LIN {X 0,Y 432.697,Z 989.03,A -85,B 0,C 180,E1 8598.502,E2 8598.502} C_VEL
LIN {X 0,Y 432.77,Z 989.03,A -85,B 0,C 180,E1 8603.648,E2 8603.648} C_VEL
LIN {X 0,Y 432.907,Z 989.03,A -85,B 0,C 180,E1 8608.477,E2 8608.477} C_VEL
LIN {X 0,Y 433.07,Z 989.297,A -85,B 0,C 180,E1 8613.186,E2 8613.186} C_VEL
LIN {X 0,Y 443.785,Z 1017.541,A -85,B 0,C 180,E1 8615.048,E2 8615.048} C_VEL
LIN {X 0,Y 445.789,Z 1028.616,A -85,B 0,C 180,E1 8615.491,E2 8615.491} C_VEL
LIN {X 0,Y 445.07,Z 1060.716,A -85,B 0,C 180,E1 8616.568,E2 8616.568} C_VEL
LIN {X 0,Y 443.495,Z 1088.889,A -85,B 0,C 180,E1 8618.283,E2 8618.283} C_VEL
LIN {X 0,Y 441.306,Z 1114.853,A -85,B 0,C 180,E1 8620.732,E2 8620.732} C_VEL
LIN {X 0,Y 439.12,Z 1136.774,A -85,B 0,C 180,E1 8623.787,E2 8623.787} C_VEL
LIN {X 0,Y 437.236,Z 1152.919,A -85,B 0,C 180,E1 8627.037,E2 8627.037} C_VEL
LIN {X 0,Y 436.045,Z 1164.999,A -85,B 0,C 180,E1 8630.715,E2 8630.715} C_VEL
LIN {X 0,Y 435.323,Z 1172.825,A -85,B 0,C 180,E1 8635.028,E2 8635.028} C_VEL
LIN {X 0,Y 435.121,Z 1174.716,A -85,B 0,C 180,E1 8638.012,E2 8638.012} C_VEL
LIN {X 0,Y 435.207,Z 1172.894,A -85,B 0,C 180,E1 8641.987,E2 8641.987} C_VEL
LIN {X 0,Y 435.483,Z 1166.041,A -85,B 0,C 180,E1 8645.966,E2 8645.966} C_VEL
LIN {X 0,Y 436.346,Z 1153.47,A -85,B 0,C 180,E1 8649.956,E2 8649.956} C_VEL
LIN {X 0,Y 437.774,Z 1136.478,A -85,B 0,C 180,E1 8653.453,E2 8653.453} C_VEL
LIN {X 0,Y 439.79,Z 1114.572,A -85,B 0,C 180,E1 8656.571,E2 8656.571} C_VEL
LIN {X 0,Y 442.047,Z 1087.996,A -85,B 0,C 180,E1 8659.181,E2 8659.181} C_VEL
LIN {X 0,Y 443.923,Z 1058.883,A -85,B 0,C 180,E1 8661.067,E2 8661.067} C_VEL
LIN {X 0,Y 445.087,Z 1027.458,A -85,B 0,C 180,E1 8662.249,E2 8662.249} C_VEL
LIN {X 0,Y 442.129,Z 1014.96,A -85,B 0,C 180,E1 8662.7,E2 8662.7} C_VEL
LIN {X 0,Y 433.211,Z 989.03,A -85,B 0,C 180,E1 8663.83,E2 8663.83} C_VEL
LIN {X 0,Y 432.895,Z 989.03,A -85,B 0,C 180,E1 8669.36,E2 8669.36} C_VEL
LIN {X 0,Y 432.823,Z 989.03,A -85,B 0,C 180,E1 8673.904,E2 8673.904} C_VEL
LIN {X 0,Y 432.669,Z 989.03,A -85,B 0,C 180,E1 8679.881,E2 8679.881} C_VEL
LIN {X 0,Y 432.821,Z 989.03,A -85,B 0,C 180,E1 8687.064,E2 8687.064} C_VEL
LIN {X 0,Y 433.004,Z 989.789,A -85,B 0,C 180,E1 8692.927,E2 8692.927} C_VEL
LIN {X 0,Y 456.109,Z 1039.383,A -85,B 0,C 180,E1 8696.121,E2 8696.121} C_VEL
LIN {X 0,Y 454.129,Z 1077.382,A -85,B 0,C 180,E1 8697.482,E2 8697.482} C_VEL
LIN {X 0,Y 450.882,Z 1111.659,A -85,B 0,C 180,E1 8699.45,E2 8699.45} C_VEL
LIN {X 0,Y 446.779,Z 1144.475,A -85,B 0,C 180,E1 8702.186,E2 8702.186} C_VEL
LIN {X 0,Y 442.832,Z 1172.505,A -85,B 0,C 180,E1 8705.44,E2 8705.44} C_VEL
LIN {X 0,Y 439.203,Z 1197.466,A -85,B 0,C 180,E1 8709.375,E2 8709.375} C_VEL
LIN {X 0,Y 436.454,Z 1218.293,A -85,B 0,C 180,E1 8713.938,E2 8713.938} C_VEL
LIN {X 0,Y 435.007,Z 1232.645,A -85,B 0,C 180,E1 8718.49,E2 8718.49} C_VEL
LIN {X 0,Y 434.441,Z 1241.786,A -85,B 0,C 180,E1 8723.013,E2 8723.013} C_VEL
LIN {X 0,Y 434.17,Z 1246.568,A -85,B 0,C 180,E1 8728.004,E2 8728.004} C_VEL
LIN {X 0,Y 434.304,Z 1246.516,A -85,B 0,C 180,E1 8731.987,E2 8731.987} C_VEL
LIN {X 0,Y 434.395,Z 1241.668,A -85,B 0,C 180,E1 8736.98,E2 8736.98} C_VEL
LIN {X 0,Y 435.171,Z 1231.159,A -85,B 0,C 180,E1 8742.005,E2 8742.005} C_VEL
LIN {X 0,Y 436.864,Z 1214.961,A -85,B 0,C 180,E1 8746.812,E2 8746.812} C_VEL
LIN {X 0,Y 439.667,Z 1194.228,A -85,B 0,C 180,E1 8751.12,E2 8751.12} C_VEL
LIN {X 0,Y 443.383,Z 1168.758,A -85,B 0,C 180,E1 8754.97,E2 8754.97} C_VEL
LIN {X 0,Y 447.385,Z 1139.749,A -85,B 0,C 180,E1 8758.175,E2 8758.175} C_VEL
LIN {X 0,Y 451.302,Z 1107.239,A -85,B 0,C 180,E1 8760.762,E2 8760.762} C_VEL
LIN {X 0,Y 454.599,Z 1071.466,A -85,B 0,C 180,E1 8762.694,E2 8762.694} C_VEL
LIN {X 0,Y 455.862,Z 1038.327,A -85,B 0,C 180,E1 8763.838,E2 8763.838} C_VEL
LIN {X 0,Y 436.175,Z 997.068,A -85,B 0,C 180,E1 8766.511,E2 8766.511} C_VEL
LIN {X 0,Y 432.88,Z 989.03,A -85,B 0,C 180,E1 8767.031,E2 8767.031} C_VEL
LIN {X 0,Y 432.718,Z 989.03,A -85,B 0,C 180,E1 8774.22,E2 8774.22} C_VEL
LIN {X 0,Y 432.769,Z 989.03,A -85,B 0,C 180,E1 8780.091,E2 8780.091} C_VEL
LIN {X 0,Y 432.886,Z 989.03,A -85,B 0,C 180,E1 8786.781,E2 8786.781} C_VEL
LIN {X 0,Y 433.033,Z 989.03,A -85,B 0,C 180,E1 8793.064,E2 8793.064} C_VEL
LIN {X 0,Y 433.316,Z 989.03,A -85,B 0,C 180,E1 8800.09,E2 8800.09} C_VEL
LIN {X 0,Y 433.537,Z 989.03,A -85,B 0,C 180,E1 8805.899,E2 8805.899} C_VEL
LIN {X 0,Y 433.62,Z 989.03,A -85,B 0,C 180,E1 8812.633,E2 8812.633} C_VEL
LIN {X 0,Y 433.826,Z 989.03,A -85,B 0,C 180,E1 8818.007,E2 8818.007} C_VEL
LIN {X 0,Y 433.765,Z 989.03,A -85,B 0,C 180,E1 8823.99,E2 8823.99} C_VEL
LIN {X 0,Y 433.535,Z 989.03,A -85,B 0,C 180,E1 8830.022,E2 8830.022} C_VEL
LIN {X 0,Y 433.346,Z 989.03,A -85,B 0,C 180,E1 8836.175,E2 8836.175} C_VEL
LIN {X 0,Y 433.179,Z 989.03,A -85,B 0,C 180,E1 8842.531,E2 8842.531} C_VEL
LIN {X 0,Y 432.896,Z 989.03,A -85,B 0,C 180,E1 8849.376,E2 8849.376} C_VEL
LIN {X 0,Y 432.837,Z 989.03,A -85,B 0,C 180,E1 8853.903,E2 8853.903} C_VEL
LIN {X 0,Y 432.775,Z 989.03,A -85,B 0,C 180,E1 8859.91,E2 8859.91} C_VEL
LIN {X 0,Y 432.855,Z 989.105,A -85,B 0,C 180,E1 8865.604,E2 8865.604} C_VEL
LIN {X 0,Y 442.678,Z 1017.502,A -85,B 0,C 180,E1 8868.683,E2 8868.683} C_VEL
LIN {X 0,Y 458.724,Z 1050.911,A -85,B 0,C 180,E1 8870.893,E2 8870.893} C_VEL
LIN {X 0,Y 460.741,Z 1053.948,A -85,B 0,C 180,E1 8871.137,E2 8871.137} C_VEL
LIN {X 0,Y 458.124,Z 1095.324,A -85,B 0,C 180,E1 8872.358,E2 8872.358} C_VEL
LIN {X 0,Y 454.341,Z 1134.437,A -85,B 0,C 180,E1 8874.243,E2 8874.243} C_VEL
LIN {X 0,Y 449.841,Z 1172.08,A -85,B 0,C 180,E1 8876.863,E2 8876.863} C_VEL
LIN {X 0,Y 446.664,Z 1196.79,A -85,B 0,C 180,E1 8879.099,E2 8879.099} C_VEL
LIN {X 0,Y 441.188,Z 1210.269,A -85,B 0,C 180,E1 8880.368,E2 8880.368} C_VEL
LIN {X 0,Y 435.677,Z 1223.042,A -85,B 0,C 180,E1 8881.762,E2 8881.762} C_VEL
LIN {X 0,Y 431.796,Z 1251.772,A -85,B 0,C 180,E1 8886.033,E2 8886.033} C_VEL
LIN {X 0,Y 428.851,Z 1276.693,A -85,B 0,C 180,E1 8891.009,E2 8891.009} C_VEL
LIN {X 0,Y 427.165,Z 1294.995,A -85,B 0,C 180,E1 8896.163,E2 8896.163} C_VEL
LIN {X 0,Y 426.423,Z 1306.284,A -85,B 0,C 180,E1 8900.841,E2 8900.841} C_VEL
LIN {X 0,Y 426.181,Z 1310.937,A -85,B 0,C 180,E1 8903.906,E2 8903.906} C_VEL
LIN {X 0,Y 426.118,Z 1314.097,A -85,B 0,C 180,E1 8907.974,E2 8907.974} C_VEL
LIN {X 0,Y 426.159,Z 1314.101,A -85,B 0,C 180,E1 8912.033,E2 8912.033} C_VEL
LIN {X 0,Y 426.297,Z 1309.951,A -85,B 0,C 180,E1 8916.886,E2 8916.886} C_VEL
LIN {X 0,Y 426.714,Z 1300.562,A -85,B 0,C 180,E1 8921.737,E2 8921.737} C_VEL
LIN {X 0,Y 427.905,Z 1286.255,A -85,B 0,C 180,E1 8926.391,E2 8926.391} C_VEL
LIN {X 0,Y 429.839,Z 1266.674,A -85,B 0,C 180,E1 8930.887,E2 8930.887} C_VEL
LIN {X 0,Y 432.863,Z 1239.391,A -85,B 0,C 180,E1 8935.454,E2 8935.454} C_VEL
LIN {X 0,Y 436.533,Z 1207.714,A -85,B 0,C 180,E1 8939.357,E2 8939.357} C_VEL
LIN {X 0,Y 440.383,Z 1171.631,A -85,B 0,C 180,E1 8942.668,E2 8942.668} C_VEL
LIN {X 0,Y 444.264,Z 1131,A -85,B 0,C 180,E1 8945.396,E2 8945.396} C_VEL
LIN {X 0,Y 447.832,Z 1087.494,A -85,B 0,C 180,E1 8947.417,E2 8947.417} C_VEL
LIN {X 0,Y 449.457,Z 1053.468,A -85,B 0,C 180,E1 8948.495,E2 8948.495} C_VEL
LIN {X 0,Y 439.336,Z 1031.663,A -85,B 0,C 180,E1 8949.877,E2 8949.877} C_VEL
LIN {X 0,Y 429.889,Z 1001.599,A -85,B 0,C 180,E1 8951.62,E2 8951.62} C_VEL
LIN {X 0,Y 424.951,Z 989.03,A -85,B 0,C 180,E1 8952.743,E2 8952.743} C_VEL
LIN {X 0,Y 424.781,Z 989.03,A -85,B 0,C 180,E1 8960.252,E2 8960.252} C_VEL
LIN {X 0,Y 424.859,Z 989.03,A -85,B 0,C 180,E1 8965.371,E2 8965.371} C_VEL
LIN {X 0,Y 425.05,Z 989.03,A -85,B 0,C 180,E1 8971.942,E2 8971.942} C_VEL
LIN {X 0,Y 425.08,Z 989.609,A -85,B 0,C 180,E1 8972.308,E2 8972.308} C_VEL
LIN {X 0,Y 435.465,Z 1014.789,A -85,B 0,C 180,E1 8974.299,E2 8974.299} C_VEL
LIN {X 0,Y 438.864,Z 1029.178,A -85,B 0,C 180,E1 8975.006,E2 8975.006} C_VEL
LIN {X 0,Y 438.027,Z 1062.901,A -85,B 0,C 180,E1 8976.168,E2 8976.168} C_VEL
LIN {X 0,Y 436.35,Z 1090.736,A -85,B 0,C 180,E1 8977.91,E2 8977.91} C_VEL
LIN {X 0,Y 434.06,Z 1116.2,A -85,B 0,C 180,E1 8980.354,E2 8980.354} C_VEL
LIN {X 0,Y 431.726,Z 1138.391,A -85,B 0,C 180,E1 8983.502,E2 8983.502} C_VEL
LIN {X 0,Y 429.681,Z 1154.456,A -85,B 0,C 180,E1 8986.805,E2 8986.805} C_VEL
LIN {X 0,Y 428.41,Z 1166.411,A -85,B 0,C 180,E1 8990.524,E2 8990.524} C_VEL
LIN {X 0,Y 427.732,Z 1173.018,A -85,B 0,C 180,E1 8993.924,E2 8993.924} C_VEL
LIN {X 0,Y 427.362,Z 1176.103,A -85,B 0,C 180,E1 8997.976,E2 8997.976} C_VEL
LIN {X 0,Y 427.447,Z 1174.222,A -85,B 0,C 180,E1 9002.023,E2 9002.023} C_VEL
LIN {X 0,Y 427.731,Z 1167.313,A -85,B 0,C 180,E1 9006.075,E2 9006.075} C_VEL
LIN {X 0,Y 428.678,Z 1154.67,A -85,B 0,C 180,E1 9010.136,E2 9010.136} C_VEL
LIN {X 0,Y 430.176,Z 1137.616,A -85,B 0,C 180,E1 9013.696,E2 9013.696} C_VEL
LIN {X 0,Y 432.314,Z 1115.636,A -85,B 0,C 180,E1 9016.866,E2 9016.866} C_VEL
LIN {X 0,Y 434.667,Z 1088.998,A -85,B 0,C 180,E1 9019.519,E2 9019.519} C_VEL
LIN {X 0,Y 436.668,Z 1058.992,A -85,B 0,C 180,E1 9021.478,E2 9021.478} C_VEL
LIN {X 0,Y 437.856,Z 1027.198,A -85,B 0,C 180,E1 9022.669,E2 9022.669} C_VEL
LIN {X 0,Y 425.204,Z 989.03,A -85,B 0,C 180,E1 9024.362,E2 9024.362} C_VEL
LIN {X 0,Y 424.94,Z 989.03,A -85,B 0,C 180,E1 9031.531,E2 9031.531} C_VEL
LIN {X 0,Y 424.741,Z 989.03,A -85,B 0,C 180,E1 9038.583,E2 9038.583} C_VEL
LIN {X 0,Y 424.87,Z 989.03,A -85,B 0,C 180,E1 9045.259,E2 9045.259} C_VEL
LIN {X 0,Y 424.987,Z 989.187,A -85,B 0,C 180,E1 9052.082,E2 9052.082} C_VEL
LIN {X 0,Y 431.957,Z 1003.724,A -85,B 0,C 180,E1 9053.108,E2 9053.108} C_VEL
LIN {X 0,Y 449.723,Z 1042.379,A -85,B 0,C 180,E1 9055.652,E2 9055.652} C_VEL
LIN {X 0,Y 447.403,Z 1079.179,A -85,B 0,C 180,E1 9056.998,E2 9056.998} C_VEL
LIN {X 0,Y 443.964,Z 1113.426,A -85,B 0,C 180,E1 9059.015,E2 9059.015} C_VEL
LIN {X 0,Y 439.582,Z 1146.278,A -85,B 0,C 180,E1 9061.83,E2 9061.83} C_VEL
LIN {X 0,Y 435.379,Z 1174.63,A -85,B 0,C 180,E1 9065.219,E2 9065.219} C_VEL
LIN {X 0,Y 431.559,Z 1199.462,A -85,B 0,C 180,E1 9069.261,E2 9069.261} C_VEL
LIN {X 0,Y 428.808,Z 1218.892,A -85,B 0,C 180,E1 9073.644,E2 9073.644} C_VEL
LIN {X 0,Y 427.245,Z 1233.244,A -85,B 0,C 180,E1 9078.278,E2 9078.278} C_VEL
LIN {X 0,Y 426.584,Z 1242.464,A -85,B 0,C 180,E1 9082.936,E2 9082.936} C_VEL
LIN {X 0,Y 426.293,Z 1247.169,A -85,B 0,C 180,E1 9087.967,E2 9087.967} C_VEL
LIN {X 0,Y 426.425,Z 1247.118,A -85,B 0,C 180,E1 9092.024,E2 9092.024} C_VEL
LIN {X 0,Y 426.543,Z 1242.349,A -85,B 0,C 180,E1 9097.056,E2 9097.056} C_VEL
LIN {X 0,Y 427.266,Z 1233.044,A -85,B 0,C 180,E1 9101.713,E2 9101.713} C_VEL
LIN {X 0,Y 428.955,Z 1218.59,A -85,B 0,C 180,E1 9106.342,E2 9106.342} C_VEL
LIN {X 0,Y 431.839,Z 1197.629,A -85,B 0,C 180,E1 9110.985,E2 9110.985} C_VEL
LIN {X 0,Y 435.654,Z 1172.61,A -85,B 0,C 180,E1 9114.972,E2 9114.972} C_VEL
LIN {X 0,Y 440.031,Z 1143.028,A -85,B 0,C 180,E1 9118.409,E2 9118.409} C_VEL
LIN {X 0,Y 444.192,Z 1110.636,A -85,B 0,C 180,E1 9121.091,E2 9121.091} C_VEL
LIN {X 0,Y 447.715,Z 1075.651,A -85,B 0,C 180,E1 9123.072,E2 9123.072} C_VEL
LIN {X 0,Y 449.208,Z 1040.792,A -85,B 0,C 180,E1 9124.351,E2 9124.351} C_VEL
LIN {X 0,Y 430.884,Z 1001.912,A -85,B 0,C 180,E1 9126.942,E2 9126.942} C_VEL
LIN {X 0,Y 424.926,Z 989.03,A -85,B 0,C 180,E1 9127.915,E2 9127.915} C_VEL
LIN {X 0,Y 424.845,Z 989.03,A -85,B 0,C 180,E1 9135.262,E2 9135.262} C_VEL
LIN {X 0,Y 424.883,Z 989.03,A -85,B 0,C 180,E1 9141.38,E2 9141.38} C_VEL
LIN {X 0,Y 424.936,Z 989.03,A -85,B 0,C 180,E1 9148.455,E2 9148.455} C_VEL
LIN {X 0,Y 425.168,Z 989.03,A -85,B 0,C 180,E1 9154.794,E2 9154.794} C_VEL
LIN {X 0,Y 425.405,Z 989.03,A -85,B 0,C 180,E1 9161.384,E2 9161.384} C_VEL
LIN {X 0,Y 425.664,Z 989.03,A -85,B 0,C 180,E1 9167.72,E2 9167.72} C_VEL
LIN {X 0,Y 425.813,Z 989.03,A -85,B 0,C 180,E1 9173.898,E2 9173.898} C_VEL
LIN {X 0,Y 426.058,Z 989.03,A -85,B 0,C 180,E1 9180,E2 9180} C_VEL
LIN {X 0,Y 425.737,Z 989.03,A -85,B 0,C 180,E1 9187.064,E2 9187.064} C_VEL
LIN {X 0,Y 425.577,Z 989.03,A -85,B 0,C 180,E1 9192.283,E2 9192.283} C_VEL
LIN {X 0,Y 425.328,Z 989.03,A -85,B 0,C 180,E1 9198.621,E2 9198.621} C_VEL
LIN {X 0,Y 425.133,Z 989.03,A -85,B 0,C 180,E1 9205.209,E2 9205.209} C_VEL
LIN {X 0,Y 424.909,Z 989.03,A -85,B 0,C 180,E1 9212.187,E2 9212.187} C_VEL
LIN {X 0,Y 424.887,Z 989.03,A -85,B 0,C 180,E1 9218.621,E2 9218.621} C_VEL
LIN {X 0,Y 424.923,Z 989.717,A -85,B 0,C 180,E1 9224.886,E2 9224.886} C_VEL
LIN {X 0,Y 434.69,Z 1016.637,A -85,B 0,C 180,E1 9227.89,E2 9227.89} C_VEL
LIN {X 0,Y 453.005,Z 1055.473,A -85,B 0,C 180,E1 9230.511,E2 9230.511} C_VEL
LIN {X 0,Y 454.078,Z 1059.186,A -85,B 0,C 180,E1 9230.7,E2 9230.7} C_VEL
LIN {X 0,Y 450.861,Z 1100.733,A -85,B 0,C 180,E1 9232.056,E2 9232.056} C_VEL
LIN {X 0,Y 446.505,Z 1141.499,A -85,B 0,C 180,E1 9234.201,E2 9234.201} C_VEL
LIN {X 0,Y 441.692,Z 1178.777,A -85,B 0,C 180,E1 9237.013,E2 9237.013} C_VEL
LIN {X 0,Y 436.921,Z 1213.948,A -85,B 0,C 180,E1 9240.629,E2 9240.629} C_VEL
LIN {X 0,Y 435.677,Z 1223.042,A -85,B 0,C 180,E1 9241.762,E2 9241.762} C_VEL
LIN {X 0,Y 430.057,Z 1235.144,A -85,B 0,C 180,E1 9243.282,E2 9243.282} C_VEL
LIN {X 0,Y 424.722,Z 1246.437,A -85,B 0,C 180,E1 9244.928,E2 9244.928} C_VEL
LIN {X 0,Y 421.591,Z 1270.624,A -85,B 0,C 180,E1 9249.578,E2 9249.578} C_VEL
LIN {X 0,Y 419.716,Z 1289.061,A -85,B 0,C 180,E1 9254.36,E2 9254.36} C_VEL
LIN {X 0,Y 418.78,Z 1301.967,A -85,B 0,C 180,E1 9259.099,E2 9259.099} C_VEL
LIN {X 0,Y 418.338,Z 1309.955,A -85,B 0,C 180,E1 9263.791,E2 9263.791} C_VEL
LIN {X 0,Y 418.241,Z 1313.389,A -85,B 0,C 180,E1 9267.936,E2 9267.936} C_VEL
LIN {X 0,Y 418.281,Z 1313.385,A -85,B 0,C 180,E1 9272.072,E2 9272.072} C_VEL
LIN {X 0,Y 418.395,Z 1309.9,A -85,B 0,C 180,E1 9276.216,E2 9276.216} C_VEL
LIN {X 0,Y 418.831,Z 1300.391,A -85,B 0,C 180,E1 9281.434,E2 9281.434} C_VEL
LIN {X 0,Y 419.957,Z 1286.383,A -85,B 0,C 180,E1 9286.174,E2 9286.174} C_VEL
LIN {X 0,Y 421.967,Z 1266.202,A -85,B 0,C 180,E1 9290.959,E2 9290.959} C_VEL
LIN {X 0,Y 424.771,Z 1241.45,A -85,B 0,C 180,E1 9295.238,E2 9295.238} C_VEL
LIN {X 0,Y 428.288,Z 1211.677,A -85,B 0,C 180,E1 9299.114,E2 9299.114} C_VEL
LIN {X 0,Y 432.282,Z 1176.111,A -85,B 0,C 180,E1 9302.591,E2 9302.591} C_VEL
LIN {X 0,Y 436.468,Z 1135.133,A -85,B 0,C 180,E1 9305.529,E2 9305.529} C_VEL
LIN {X 0,Y 440.479,Z 1090.079,A -85,B 0,C 180,E1 9307.767,E2 9307.767} C_VEL
LIN {X 0,Y 442.462,Z 1056.367,A -85,B 0,C 180,E1 9308.923,E2 9308.923} C_VEL
LIN {X 0,Y 432.925,Z 1034.002,A -85,B 0,C 180,E1 9310.416,E2 9310.416} C_VEL
LIN {X 0,Y 423.891,Z 1004.177,A -85,B 0,C 180,E1 9312.262,E2 9312.262} C_VEL
LIN {X 0,Y 418.544,Z 993.693,A -85,B 0,C 180,E1 9313.357,E2 9313.357} C_VEL
LIN {X 0,Y 416.956,Z 989.03,A -85,B 0,C 180,E1 9313.91,E2 9313.91} C_VEL
LIN {X 0,Y 416.829,Z 989.03,A -85,B 0,C 180,E1 9319.494,E2 9319.494} C_VEL
LIN {X 0,Y 416.916,Z 989.03,A -85,B 0,C 180,E1 9326.363,E2 9326.363} C_VEL
LIN {X 0,Y 417.138,Z 989.03,A -85,B 0,C 180,E1 9331.219,E2 9331.219} C_VEL
LIN {X 0,Y 427.512,Z 1013.324,A -85,B 0,C 180,E1 9333.524,E2 9333.524} C_VEL
LIN {X 0,Y 432.04,Z 1030.019,A -85,B 0,C 180,E1 9334.495,E2 9334.495} C_VEL
LIN {X 0,Y 431.091,Z 1064.164,A -85,B 0,C 180,E1 9335.697,E2 9335.697} C_VEL
LIN {X 0,Y 429.277,Z 1092.763,A -85,B 0,C 180,E1 9337.526,E2 9337.526} C_VEL
LIN {X 0,Y 426.758,Z 1118.671,A -85,B 0,C 180,E1 9340.089,E2 9340.089} C_VEL
LIN {X 0,Y 424.327,Z 1140.066,A -85,B 0,C 180,E1 9343.206,E2 9343.206} C_VEL
LIN {X 0,Y 422.143,Z 1156.036,A -85,B 0,C 180,E1 9346.565,E2 9346.565} C_VEL
LIN {X 0,Y 420.754,Z 1167.929,A -85,B 0,C 180,E1 9350.35,E2 9350.35} C_VEL
LIN {X 0,Y 420.03,Z 1174.471,A -85,B 0,C 180,E1 9353.813,E2 9353.813} C_VEL
LIN {X 0,Y 419.606,Z 1177.5,A -85,B 0,C 180,E1 9357.939,E2 9357.939} C_VEL
LIN {X 0,Y 419.679,Z 1175.549,A -85,B 0,C 180,E1 9362.06,E2 9362.06} C_VEL
LIN {X 0,Y 419.988,Z 1168.561,A -85,B 0,C 180,E1 9366.187,E2 9366.187} C_VEL
LIN {X 0,Y 420.994,Z 1155.832,A -85,B 0,C 180,E1 9370.323,E2 9370.323} C_VEL
LIN {X 0,Y 422.574,Z 1138.687,A -85,B 0,C 180,E1 9373.947,E2 9373.947} C_VEL
LIN {X 0,Y 424.921,Z 1115.581,A -85,B 0,C 180,E1 9377.301,E2 9377.301} C_VEL
LIN {X 0,Y 427.441,Z 1088.267,A -85,B 0,C 180,E1 9379.997,E2 9379.997} C_VEL
LIN {X 0,Y 429.389,Z 1059.763,A -85,B 0,C 180,E1 9381.861,E2 9381.861} C_VEL
LIN {X 0,Y 430.389,Z 1026.985,A -85,B 0,C 180,E1 9383.107,E2 9383.107} C_VEL
LIN {X 0,Y 417.283,Z 989.03,A -85,B 0,C 180,E1 9384.893,E2 9384.893} C_VEL
LIN {X 0,Y 417.025,Z 989.03,A -85,B 0,C 180,E1 9390.435,E2 9390.435} C_VEL
LIN {X 0,Y 416.847,Z 989.03,A -85,B 0,C 180,E1 9397.202,E2 9397.202} C_VEL
LIN {X 0,Y 416.84,Z 989.03,A -85,B 0,C 180,E1 9403.605,E2 9403.605} C_VEL
LIN {X 0,Y 416.976,Z 989.03,A -85,B 0,C 180,E1 9410.496,E2 9410.496} C_VEL
LIN {X 0,Y 417.012,Z 989.033,A -85,B 0,C 180,E1 9411.209,E2 9411.209} C_VEL
LIN {X 0,Y 421.339,Z 998.671,A -85,B 0,C 180,E1 9411.893,E2 9411.893} C_VEL
LIN {X 0,Y 441.202,Z 1039.657,A -85,B 0,C 180,E1 9414.786,E2 9414.786} C_VEL
LIN {X 0,Y 443.045,Z 1046.799,A -85,B 0,C 180,E1 9415.186,E2 9415.186} C_VEL
LIN {X 0,Y 440.312,Z 1084.785,A -85,B 0,C 180,E1 9416.679,E2 9416.679} C_VEL
LIN {X 0,Y 436.489,Z 1119.573,A -85,B 0,C 180,E1 9418.902,E2 9418.902} C_VEL
LIN {X 0,Y 432.046,Z 1150.522,A -85,B 0,C 180,E1 9421.72,E2 9421.72} C_VEL
LIN {X 0,Y 427.643,Z 1178.421,A -85,B 0,C 180,E1 9425.222,E2 9425.222} C_VEL
LIN {X 0,Y 423.67,Z 1202.649,A -85,B 0,C 180,E1 9429.402,E2 9429.402} C_VEL
LIN {X 0,Y 420.924,Z 1221.353,A -85,B 0,C 180,E1 9433.864,E2 9433.864} C_VEL
LIN {X 0,Y 419.347,Z 1235.118,A -85,B 0,C 180,E1 9438.58,E2 9438.58} C_VEL
LIN {X 0,Y 418.641,Z 1244.422,A -85,B 0,C 180,E1 9443.788,E2 9443.788} C_VEL
LIN {X 0,Y 418.415,Z 1247.77,A -85,B 0,C 180,E1 9447.929,E2 9447.929} C_VEL
LIN {X 0,Y 418.545,Z 1247.72,A -85,B 0,C 180,E1 9452.062,E2 9452.062} C_VEL
LIN {X 0,Y 418.678,Z 1243.217,A -85,B 0,C 180,E1 9457.002,E2 9457.002} C_VEL
LIN {X 0,Y 419.504,Z 1233.648,A -85,B 0,C 180,E1 9461.933,E2 9461.933} C_VEL
LIN {X 0,Y 421.281,Z 1219.199,A -85,B 0,C 180,E1 9466.648,E2 9466.648} C_VEL
LIN {X 0,Y 424.36,Z 1198.426,A -85,B 0,C 180,E1 9471.335,E2 9471.335} C_VEL
LIN {X 0,Y 428.369,Z 1173.656,A -85,B 0,C 180,E1 9475.359,E2 9475.359} C_VEL
LIN {X 0,Y 433.085,Z 1143.62,A -85,B 0,C 180,E1 9478.908,E2 9478.908} C_VEL
LIN {X 0,Y 437.471,Z 1111.065,A -85,B 0,C 180,E1 9481.635,E2 9481.635} C_VEL
LIN {X 0,Y 441.144,Z 1075.926,A -85,B 0,C 180,E1 9483.645,E2 9483.645} C_VEL
LIN {X 0,Y 442.733,Z 1043.418,A -85,B 0,C 180,E1 9484.858,E2 9484.858} C_VEL
LIN {X 0,Y 424.334,Z 1004.19,A -85,B 0,C 180,E1 9487.572,E2 9487.572} C_VEL
LIN {X 0,Y 417.022,Z 990.228,A -85,B 0,C 180,E1 9488.665,E2 9488.665} C_VEL
LIN {X 0,Y 416.949,Z 989.03,A -85,B 0,C 180,E1 9488.725,E2 9488.725} C_VEL
LIN {X 0,Y 416.877,Z 989.03,A -85,B 0,C 180,E1 9496.378,E2 9496.378} C_VEL
LIN {X 0,Y 417.014,Z 989.03,A -85,B 0,C 180,E1 9502.754,E2 9502.754} C_VEL
LIN {X 0,Y 417.058,Z 989.03,A -85,B 0,C 180,E1 9510.265,E2 9510.265} C_VEL
LIN {X 0,Y 417.304,Z 989.03,A -85,B 0,C 180,E1 9516.563,E2 9516.563} C_VEL
LIN {X 0,Y 417.566,Z 989.03,A -85,B 0,C 180,E1 9523.197,E2 9523.197} C_VEL
LIN {X 0,Y 417.761,Z 989.03,A -85,B 0,C 180,E1 9529.596,E2 9529.596} C_VEL
LIN {X 0,Y 417.998,Z 989.03,A -85,B 0,C 180,E1 9535.86,E2 9535.86} C_VEL
LIN {X 0,Y 418.182,Z 989.03,A -85,B 0,C 180,E1 9542.068,E2 9542.068} C_VEL
LIN {X 0,Y 417.79,Z 989.03,A -85,B 0,C 180,E1 9548.307,E2 9548.307} C_VEL
LIN {X 0,Y 417.539,Z 989.03,A -85,B 0,C 180,E1 9554.654,E2 9554.654} C_VEL
LIN {X 0,Y 417.337,Z 989.03,A -85,B 0,C 180,E1 9561.197,E2 9561.197} C_VEL
LIN {X 0,Y 417.067,Z 989.03,A -85,B 0,C 180,E1 9568.057,E2 9568.057} C_VEL
LIN {X 0,Y 416.946,Z 989.03,A -85,B 0,C 180,E1 9575.384,E2 9575.384} C_VEL
LIN {X 0,Y 416.921,Z 989.03,A -85,B 0,C 180,E1 9580.653,E2 9580.653} C_VEL
LIN {X 0,Y 416.937,Z 989.221,A -85,B 0,C 180,E1 9584.043,E2 9584.043} C_VEL
LIN {X 0,Y 426.396,Z 1015.45,A -85,B 0,C 180,E1 9587.037,E2 9587.037} C_VEL
LIN {X 0,Y 447.39,Z 1061.599,A -85,B 0,C 180,E1 9590.201,E2 9590.201} C_VEL
LIN {X 0,Y 443.922,Z 1102.643,A -85,B 0,C 180,E1 9591.607,E2 9591.607} C_VEL
LIN {X 0,Y 439.459,Z 1141.866,A -85,B 0,C 180,E1 9593.742,E2 9593.742} C_VEL
LIN {X 0,Y 434.489,Z 1178.285,A -85,B 0,C 180,E1 9596.555,E2 9596.555} C_VEL
LIN {X 0,Y 429.614,Z 1212.439,A -85,B 0,C 180,E1 9600.116,E2 9600.116} C_VEL
LIN {X 0,Y 425.114,Z 1243.426,A -85,B 0,C 180,E1 9604.439,E2 9604.439} C_VEL
LIN {X 0,Y 424.722,Z 1246.437,A -85,B 0,C 180,E1 9604.928,E2 9604.928} C_VEL
LIN {X 0,Y 421.237,Z 1254.435,A -85,B 0,C 180,E1 9606.259,E2 9606.259} C_VEL
LIN {X 0,Y 414.479,Z 1265.411,A -85,B 0,C 180,E1 9608.334,E2 9608.334} C_VEL
LIN {X 0,Y 414.243,Z 1266.576,A -85,B 0,C 180,E1 9608.588,E2 9608.588} C_VEL
LIN {X 0,Y 412.038,Z 1285.97,A -85,B 0,C 180,E1 9613.515,E2 9613.515} C_VEL
LIN {X 0,Y 410.953,Z 1300.769,A -85,B 0,C 180,E1 9618.889,E2 9618.889} C_VEL
LIN {X 0,Y 410.522,Z 1308.819,A -85,B 0,C 180,E1 9623.673,E2 9623.673} C_VEL
LIN {X 0,Y 410.418,Z 1312.221,A -85,B 0,C 180,E1 9627.897,E2 9627.897} C_VEL
LIN {X 0,Y 410.461,Z 1312.183,A -85,B 0,C 180,E1 9632.111,E2 9632.111} C_VEL
LIN {X 0,Y 410.608,Z 1307.489,A -85,B 0,C 180,E1 9637.149,E2 9637.149} C_VEL
LIN {X 0,Y 411.14,Z 1297.635,A -85,B 0,C 180,E1 9642.188,E2 9642.188} C_VEL
LIN {X 0,Y 412.484,Z 1281.775,A -85,B 0,C 180,E1 9647.293,E2 9647.293} C_VEL
LIN {X 0,Y 414.732,Z 1259.876,A -85,B 0,C 180,E1 9652.184,E2 9652.184} C_VEL
LIN {X 0,Y 417.912,Z 1233.251,A -85,B 0,C 180,E1 9656.546,E2 9656.546} C_VEL
LIN {X 0,Y 421.889,Z 1200.631,A -85,B 0,C 180,E1 9660.536,E2 9660.536} C_VEL
LIN {X 0,Y 426.217,Z 1163.51,A -85,B 0,C 180,E1 9663.924,E2 9663.924} C_VEL
LIN {X 0,Y 430.599,Z 1121.292,A -85,B 0,C 180,E1 9666.729,E2 9666.729} C_VEL
LIN {X 0,Y 434.662,Z 1077.509,A -85,B 0,C 180,E1 9668.725,E2 9668.725} C_VEL
LIN {X 0,Y 435.59,Z 1059.318,A -85,B 0,C 180,E1 9669.372,E2 9669.372} C_VEL
LIN {X 0,Y 426.067,Z 1034.638,A -85,B 0,C 180,E1 9671.089,E2 9671.089} C_VEL
LIN {X 0,Y 418.545,Z 1008.074,A -85,B 0,C 180,E1 9672.845,E2 9672.845} C_VEL
LIN {X 0,Y 411.617,Z 994.871,A -85,B 0,C 180,E1 9674.428,E2 9674.428} C_VEL
LIN {X 0,Y 409.087,Z 989.937,A -85,B 0,C 180,E1 9675.125,E2 9675.125} C_VEL
LIN {X 0,Y 409.027,Z 989.03,A -85,B 0,C 180,E1 9675.498,E2 9675.498} C_VEL
LIN {X 0,Y 408.861,Z 989.03,A -85,B 0,C 180,E1 9681.141,E2 9681.141} C_VEL
LIN {X 0,Y 409.052,Z 989.03,A -85,B 0,C 180,E1 9688.057,E2 9688.057} C_VEL
LIN {X 0,Y 409.23,Z 989.101,A -85,B 0,C 180,E1 9689.961,E2 9689.961} C_VEL
LIN {X 0,Y 411.824,Z 994.878,A -85,B 0,C 180,E1 9690.757,E2 9690.757} C_VEL
LIN {X 0,Y 420.714,Z 1014.829,A -85,B 0,C 180,E1 9692.884,E2 9692.884} C_VEL
LIN {X 0,Y 425.328,Z 1031.966,A -85,B 0,C 180,E1 9693.984,E2 9693.984} C_VEL
LIN {X 0,Y 424.181,Z 1066.846,A -85,B 0,C 180,E1 9695.275,E2 9695.275} C_VEL
LIN {X 0,Y 422.248,Z 1094.926,A -85,B 0,C 180,E1 9697.13,E2 9697.13} C_VEL
LIN {X 0,Y 419.564,Z 1120.668,A -85,B 0,C 180,E1 9699.743,E2 9699.743} C_VEL
LIN {X 0,Y 416.971,Z 1141.781,A -85,B 0,C 180,E1 9702.9,E2 9702.9} C_VEL
LIN {X 0,Y 414.628,Z 1157.668,A -85,B 0,C 180,E1 9706.316,E2 9706.316} C_VEL
LIN {X 0,Y 412.987,Z 1170.551,A -85,B 0,C 180,E1 9710.627,E2 9710.627} C_VEL
LIN {X 0,Y 412.098,Z 1177.173,A -85,B 0,C 180,E1 9714.747,E2 9714.747} C_VEL
LIN {X 0,Y 411.848,Z 1178.901,A -85,B 0,C 180,E1 9717.9,E2 9717.9} C_VEL
LIN {X 0,Y 411.917,Z 1176.875,A -85,B 0,C 180,E1 9722.099,E2 9722.099} C_VEL
LIN {X 0,Y 412.236,Z 1169.807,A -85,B 0,C 180,E1 9726.304,E2 9726.304} C_VEL
LIN {X 0,Y 413.311,Z 1156.991,A -85,B 0,C 180,E1 9730.517,E2 9730.517} C_VEL
LIN {X 0,Y 415.001,Z 1139.756,A -85,B 0,C 180,E1 9734.207,E2 9734.207} C_VEL
LIN {X 0,Y 417.336,Z 1117.605,A -85,B 0,C 180,E1 9737.49,E2 9737.49} C_VEL
LIN {X 0,Y 419.927,Z 1090.766,A -85,B 0,C 180,E1 9740.234,E2 9740.234} C_VEL
LIN {X 0,Y 422.113,Z 1060.656,A -85,B 0,C 180,E1 9742.251,E2 9742.251} C_VEL
LIN {X 0,Y 422.891,Z 1028.003,A -85,B 0,C 180,E1 9743.532,E2 9743.532} C_VEL
LIN {X 0,Y 409.302,Z 989.03,A -85,B 0,C 180,E1 9745.437,E2 9745.437} C_VEL
LIN {X 0,Y 408.989,Z 989.03,A -85,B 0,C 180,E1 9751.929,E2 9751.929} C_VEL
LIN {X 0,Y 408.83,Z 989.03,A -85,B 0,C 180,E1 9758.862,E2 9758.862} C_VEL
LIN {X 0,Y 408.881,Z 989.03,A -85,B 0,C 180,E1 9765.468,E2 9765.468} C_VEL
LIN {X 0,Y 409.085,Z 989.03,A -85,B 0,C 180,E1 9770.265,E2 9770.265} C_VEL
LIN {X 0,Y 413.754,Z 999.171,A -85,B 0,C 180,E1 9771.064,E2 9771.064} C_VEL
LIN {X 0,Y 433.445,Z 1039.137,A -85,B 0,C 180,E1 9774.031,E2 9774.031} C_VEL
LIN {X 0,Y 436.594,Z 1047.61,A -85,B 0,C 180,E1 9774.606,E2 9774.606} C_VEL
LIN {X 0,Y 433.738,Z 1085.338,A -85,B 0,C 180,E1 9776.106,E2 9776.106} C_VEL
LIN {X 0,Y 429.748,Z 1120.157,A -85,B 0,C 180,E1 9778.359,E2 9778.359} C_VEL
LIN {X 0,Y 425.086,Z 1151.106,A -85,B 0,C 180,E1 9781.214,E2 9781.214} C_VEL
LIN {X 0,Y 420.414,Z 1179.016,A -85,B 0,C 180,E1 9784.766,E2 9784.766} C_VEL
LIN {X 0,Y 416.215,Z 1203.249,A -85,B 0,C 180,E1 9789.016,E2 9789.016} C_VEL
LIN {X 0,Y 413.252,Z 1221.957,A -85,B 0,C 180,E1 9793.556,E2 9793.556} C_VEL
LIN {X 0,Y 411.558,Z 1235.721,A -85,B 0,C 180,E1 9798.361,E2 9798.361} C_VEL
LIN {X 0,Y 410.801,Z 1245.023,A -85,B 0,C 180,E1 9803.669,E2 9803.669} C_VEL
LIN {X 0,Y 410.538,Z 1248.371,A -85,B 0,C 180,E1 9807.889,E2 9807.889} C_VEL
LIN {X 0,Y 410.666,Z 1248.322,A -85,B 0,C 180,E1 9812.102,E2 9812.102} C_VEL
LIN {X 0,Y 410.852,Z 1243.424,A -85,B 0,C 180,E1 9817.422,E2 9817.422} C_VEL
LIN {X 0,Y 411.875,Z 1232.976,A -85,B 0,C 180,E1 9822.695,E2 9822.695} C_VEL
LIN {X 0,Y 413.806,Z 1218.02,A -85,B 0,C 180,E1 9827.452,E2 9827.452} C_VEL
LIN {X 0,Y 417.248,Z 1197.053,A -85,B 0,C 180,E1 9832.112,E2 9832.112} C_VEL
LIN {X 0,Y 421.785,Z 1171.065,A -85,B 0,C 180,E1 9836.272,E2 9836.272} C_VEL
LIN {X 0,Y 426.582,Z 1141.526,A -85,B 0,C 180,E1 9839.682,E2 9839.682} C_VEL
LIN {X 0,Y 431.125,Z 1109.058,A -85,B 0,C 180,E1 9842.365,E2 9842.365} C_VEL
LIN {X 0,Y 434.912,Z 1073.188,A -85,B 0,C 180,E1 9844.372,E2 9844.372} C_VEL
LIN {X 0,Y 436.139,Z 1045.874,A -85,B 0,C 180,E1 9845.4,E2 9845.4} C_VEL
LIN {X 0,Y 419.161,Z 1009.204,A -85,B 0,C 180,E1 9848.019,E2 9848.019} C_VEL
LIN {X 0,Y 409.033,Z 989.762,A -85,B 0,C 180,E1 9849.591,E2 9849.591} C_VEL
LIN {X 0,Y 408.86,Z 989.03,A -85,B 0,C 180,E1 9855.476,E2 9855.476} C_VEL
LIN {X 0,Y 408.967,Z 989.03,A -85,B 0,C 180,E1 9861.154,E2 9861.154} C_VEL
LIN {X 0,Y 409.016,Z 989.03,A -85,B 0,C 180,E1 9866.401,E2 9866.401} C_VEL
LIN {X 0,Y 409.211,Z 989.03,A -85,B 0,C 180,E1 9873.737,E2 9873.737} C_VEL
LIN {X 0,Y 409.512,Z 989.03,A -85,B 0,C 180,E1 9880.633,E2 9880.633} C_VEL
LIN {X 0,Y 409.813,Z 989.03,A -85,B 0,C 180,E1 9887.237,E2 9887.237} C_VEL
LIN {X 0,Y 410.023,Z 989.03,A -85,B 0,C 180,E1 9893.662,E2 9893.662} C_VEL
LIN {X 0,Y 410.262,Z 989.03,A -85,B 0,C 180,E1 9900,E2 9900} C_VEL
LIN {X 0,Y 410.008,Z 989.03,A -85,B 0,C 180,E1 9906.446,E2 9906.446} C_VEL
LIN {X 0,Y 409.73,Z 989.03,A -85,B 0,C 180,E1 9912.766,E2 9912.766} C_VEL
LIN {X 0,Y 409.442,Z 989.03,A -85,B 0,C 180,E1 9919.371,E2 9919.371} C_VEL
LIN {X 0,Y 409.193,Z 989.03,A -85,B 0,C 180,E1 9926.265,E2 9926.265} C_VEL
LIN {X 0,Y 409.01,Z 989.03,A -85,B 0,C 180,E1 9933.6,E2 9933.6} C_VEL
LIN {X 0,Y 408.949,Z 989.03,A -85,B 0,C 180,E1 9939.209,E2 9939.209} C_VEL
LIN {X 0,Y 409.02,Z 989.704,A -85,B 0,C 180,E1 9943.28,E2 9943.28} C_VEL
LIN {X 0,Y 418.039,Z 1014.15,A -85,B 0,C 180,E1 9946.15,E2 9946.15} C_VEL
LIN {X 0,Y 440.686,Z 1064.356,A -85,B 0,C 180,E1 9949.7,E2 9949.7} C_VEL
LIN {X 0,Y 436.753,Z 1106.23,A -85,B 0,C 180,E1 9951.232,E2 9951.232} C_VEL
LIN {X 0,Y 431.801,Z 1146.316,A -85,B 0,C 180,E1 9953.555,E2 9953.555} C_VEL
LIN {X 0,Y 426.425,Z 1183.67,A -85,B 0,C 180,E1 9956.632,E2 9956.632} C_VEL
LIN {X 0,Y 421.183,Z 1218.097,A -85,B 0,C 180,E1 9960.488,E2 9960.488} C_VEL
LIN {X 0,Y 416.831,Z 1247.664,A -85,B 0,C 180,E1 9964.924,E2 9964.924} C_VEL
LIN {X 0,Y 414.243,Z 1266.576,A -85,B 0,C 180,E1 9968.588,E2 9968.588} C_VEL
LIN {X 0,Y 409.308,Z 1275.337,A -85,B 0,C 180,E1 9970.586,E2 9970.586} C_VEL
LIN {X 0,Y 404.443,Z 1283.093,A -85,B 0,C 180,E1 9972.707,E2 9972.707} C_VEL
LIN {X 0,Y 403.21,Z 1296.992,A -85,B 0,C 180,E1 9977.577,E2 9977.577} C_VEL
LIN {X 0,Y 402.768,Z 1306.662,A -85,B 0,C 180,E1 9982.76,E2 9982.76} C_VEL
LIN {X 0,Y 402.595,Z 1311.049,A -85,B 0,C 180,E1 9987.856,E2 9987.856} C_VEL
LIN {X 0,Y 402.641,Z 1310.981,A -85,B 0,C 180,E1 9992.152,E2 9992.152} C_VEL
LIN {X 0,Y 402.789,Z 1306.182,A -85,B 0,C 180,E1 9997.288,E2 9997.288} C_VEL
LIN {X 0,Y 403.35,Z 1296.134,A -85,B 0,C 180,E1 10002.427,E2 10002.427} C_VEL
LIN {X 0,Y 404.736,Z 1279.974,A -85,B 0,C 180,E1 10007.635,E2 10007.635} C_VEL
LIN {X 0,Y 407.112,Z 1257.617,A -85,B 0,C 180,E1 10012.64,E2 10012.64} C_VEL
LIN {X 0,Y 410.4,Z 1230.76,A -85,B 0,C 180,E1 10017.044,E2 10017.044} C_VEL
LIN {X 0,Y 414.548,Z 1197.916,A -85,B 0,C 180,E1 10021.078,E2 10021.078} C_VEL
LIN {X 0,Y 419.209,Z 1159.265,A -85,B 0,C 180,E1 10024.609,E2 10024.609} C_VEL
LIN {X 0,Y 423.947,Z 1116.521,A -85,B 0,C 180,E1 10027.438,E2 10027.438} C_VEL
LIN {X 0,Y 428.18,Z 1074.117,A -85,B 0,C 180,E1 10029.379,E2 10029.379} C_VEL
LIN {X 0,Y 428.668,Z 1062.031,A -85,B 0,C 180,E1 10029.848,E2 10029.848} C_VEL
LIN {X 0,Y 419.641,Z 1036.152,A -85,B 0,C 180,E1 10031.744,E2 10031.744} C_VEL
LIN {X 0,Y 413.275,Z 1011.929,A -85,B 0,C 180,E1 10033.474,E2 10033.474} C_VEL
LIN {X 0,Y 406.735,Z 999.865,A -85,B 0,C 180,E1 10035.105,E2 10035.105} C_VEL
LIN {X 0,Y 403.745,Z 994.989,A -85,B 0,C 180,E1 10035.994,E2 10035.994} C_VEL
LIN {X 0,Y 400.991,Z 989.816,A -85,B 0,C 180,E1 10037.011,E2 10037.011} C_VEL
LIN {X 0,Y 400.946,Z 989.03,A -85,B 0,C 180,E1 10042.975,E2 10042.975} C_VEL
LIN {X 0,Y 401.171,Z 989.16,A -85,B 0,C 180,E1 10048.224,E2 10048.224} C_VEL
LIN {X 0,Y 403.725,Z 994.768,A -85,B 0,C 180,E1 10049.291,E2 10049.291} C_VEL
LIN {X 0,Y 410.369,Z 1007.776,A -85,B 0,C 180,E1 10051.264,E2 10051.264} C_VEL
LIN {X 0,Y 417.344,Z 1026.752,A -85,B 0,C 180,E1 10053.01,E2 10053.01} C_VEL
LIN {X 0,Y 418.606,Z 1036.102,A -85,B 0,C 180,E1 10053.507,E2 10053.507} C_VEL
LIN {X 0,Y 417.333,Z 1069.762,A -85,B 0,C 180,E1 10054.838,E2 10054.838} C_VEL
LIN {X 0,Y 415.239,Z 1097.241,A -85,B 0,C 180,E1 10056.722,E2 10056.722} C_VEL
LIN {X 0,Y 412.495,Z 1121.863,A -85,B 0,C 180,E1 10059.277,E2 10059.277} C_VEL
LIN {X 0,Y 409.649,Z 1143.587,A -85,B 0,C 180,E1 10062.585,E2 10062.585} C_VEL
LIN {X 0,Y 407.123,Z 1159.333,A -85,B 0,C 180,E1 10066.059,E2 10066.059} C_VEL
LIN {X 0,Y 405.537,Z 1170.761,A -85,B 0,C 180,E1 10069.866,E2 10069.866} C_VEL
LIN {X 0,Y 404.627,Z 1177.444,A -85,B 0,C 180,E1 10073.576,E2 10073.576} C_VEL
LIN {X 0,Y 404.088,Z 1180.318,A -85,B 0,C 180,E1 10077.86,E2 10077.86} C_VEL
LIN {X 0,Y 404.146,Z 1178.205,A -85,B 0,C 180,E1 10082.139,E2 10082.139} C_VEL
LIN {X 0,Y 404.473,Z 1171.051,A -85,B 0,C 180,E1 10086.426,E2 10086.426} C_VEL
LIN {X 0,Y 405.626,Z 1158.131,A -85,B 0,C 180,E1 10090.719,E2 10090.719} C_VEL
LIN {X 0,Y 407.597,Z 1139.274,A -85,B 0,C 180,E1 10094.744,E2 10094.744} C_VEL
LIN {X 0,Y 410.138,Z 1116.319,A -85,B 0,C 180,E1 10098.084,E2 10098.084} C_VEL
LIN {X 0,Y 412.764,Z 1089.149,A -85,B 0,C 180,E1 10100.806,E2 10100.806} C_VEL
LIN {X 0,Y 414.973,Z 1059.364,A -85,B 0,C 180,E1 10102.76,E2 10102.76} C_VEL
LIN {X 0,Y 415.627,Z 1029.66,A -85,B 0,C 180,E1 10103.935,E2 10103.935} C_VEL
LIN {X 0,Y 401.339,Z 989.03,A -85,B 0,C 180,E1 10105.957,E2 10105.957} C_VEL
LIN {X 0,Y 401.111,Z 989.03,A -85,B 0,C 180,E1 10111.78,E2 10111.78} C_VEL
LIN {X 0,Y 400.866,Z 989.03,A -85,B 0,C 180,E1 10117.757,E2 10117.757} C_VEL
LIN {X 0,Y 400.95,Z 989.03,A -85,B 0,C 180,E1 10124.342,E2 10124.342} C_VEL
LIN {X 0,Y 401.202,Z 989.63,A -85,B 0,C 180,E1 10129.358,E2 10129.358} C_VEL
LIN {X 0,Y 425.243,Z 1037.607,A -85,B 0,C 180,E1 10133.169,E2 10133.169} C_VEL
LIN {X 0,Y 430.054,Z 1051.41,A -85,B 0,C 180,E1 10134.095,E2 10134.095} C_VEL
LIN {X 0,Y 426.916,Z 1088.572,A -85,B 0,C 180,E1 10135.664,E2 10135.664} C_VEL
LIN {X 0,Y 422.755,Z 1122.704,A -85,B 0,C 180,E1 10137.954,E2 10137.954} C_VEL
LIN {X 0,Y 417.747,Z 1154.132,A -85,B 0,C 180,E1 10140.956,E2 10140.956} C_VEL
LIN {X 0,Y 412.893,Z 1181.331,A -85,B 0,C 180,E1 10144.563,E2 10144.563} C_VEL
LIN {X 0,Y 408.542,Z 1205.122,A -85,B 0,C 180,E1 10148.887,E2 10148.887} C_VEL
LIN {X 0,Y 405.38,Z 1224.418,A -85,B 0,C 180,E1 10153.784,E2 10153.784} C_VEL
LIN {X 0,Y 403.662,Z 1237.551,A -85,B 0,C 180,E1 10158.677,E2 10158.677} C_VEL
LIN {X 0,Y 402.948,Z 1245.625,A -85,B 0,C 180,E1 10163.545,E2 10163.545} C_VEL
LIN {X 0,Y 402.683,Z 1248.97,A -85,B 0,C 180,E1 10167.848,E2 10167.848} C_VEL
LIN {X 0,Y 402.8,Z 1248.923,A -85,B 0,C 180,E1 10172.143,E2 10172.143} C_VEL
LIN {X 0,Y 403.023,Z 1244.026,A -85,B 0,C 180,E1 10177.567,E2 10177.567} C_VEL
LIN {X 0,Y 404.131,Z 1233.581,A -85,B 0,C 180,E1 10182.942,E2 10182.942} C_VEL
LIN {X 0,Y 406.404,Z 1217.255,A -85,B 0,C 180,E1 10188.15,E2 10188.15} C_VEL
LIN {X 0,Y 410.002,Z 1196.746,A -85,B 0,C 180,E1 10192.711,E2 10192.711} C_VEL
LIN {X 0,Y 414.904,Z 1170.296,A -85,B 0,C 180,E1 10196.94,E2 10196.94} C_VEL
LIN {X 0,Y 419.899,Z 1140.913,A -85,B 0,C 180,E1 10200.337,E2 10200.337} C_VEL
LIN {X 0,Y 424.605,Z 1108.551,A -85,B 0,C 180,E1 10203.015,E2 10203.015} C_VEL
LIN {X 0,Y 428.548,Z 1072.208,A -85,B 0,C 180,E1 10205.032,E2 10205.032} C_VEL
LIN {X 0,Y 429.783,Z 1048.83,A -85,B 0,C 180,E1 10205.923,E2 10205.923} C_VEL
LIN {X 0,Y 414.725,Z 1015.704,A -85,B 0,C 180,E1 10208.365,E2 10208.365} C_VEL
LIN {X 0,Y 401.242,Z 990.938,A -85,B 0,C 180,E1 10210.504,E2 10210.504} C_VEL
LIN {X 0,Y 400.995,Z 989.03,A -85,B 0,C 180,E1 10210.696,E2 10210.696} C_VEL
LIN {X 0,Y 400.968,Z 989.03,A -85,B 0,C 180,E1 10217.361,E2 10217.361} C_VEL
LIN {X 0,Y 401.017,Z 989.03,A -85,B 0,C 180,E1 10222.984,E2 10222.984} C_VEL
LIN {X 0,Y 401.097,Z 989.03,A -85,B 0,C 180,E1 10229.912,E2 10229.912} C_VEL
LIN {X 0,Y 401.36,Z 989.03,A -85,B 0,C 180,E1 10235.572,E2 10235.572} C_VEL
LIN {X 0,Y 401.673,Z 989.03,A -85,B 0,C 180,E1 10242.511,E2 10242.511} C_VEL
LIN {X 0,Y 401.918,Z 989.03,A -85,B 0,C 180,E1 10249.181,E2 10249.181} C_VEL
LIN {X 0,Y 402.188,Z 989.03,A -85,B 0,C 180,E1 10255.697,E2 10255.697} C_VEL
LIN {X 0,Y 402.383,Z 989.03,A -85,B 0,C 180,E1 10262.15,E2 10262.15} C_VEL
LIN {X 0,Y 401.958,Z 989.03,A -85,B 0,C 180,E1 10268.637,E2 10268.637} C_VEL
LIN {X 0,Y 401.688,Z 989.03,A -85,B 0,C 180,E1 10275.246,E2 10275.246} C_VEL
LIN {X 0,Y 401.427,Z 989.03,A -85,B 0,C 180,E1 10282.08,E2 10282.08} C_VEL
LIN {X 0,Y 401.12,Z 989.03,A -85,B 0,C 180,E1 10289.278,E2 10289.278} C_VEL
LIN {X 0,Y 401.076,Z 989.03,A -85,B 0,C 180,E1 10294.357,E2 10294.357} C_VEL
LIN {X 0,Y 400.965,Z 989.03,A -85,B 0,C 180,E1 10301.181,E2 10301.181} C_VEL
LIN {X 0,Y 401.038,Z 989.64,A -85,B 0,C 180,E1 10302.437,E2 10302.437} C_VEL
LIN {X 0,Y 409.773,Z 1013.046,A -85,B 0,C 180,E1 10305.248,E2 10305.248} C_VEL
LIN {X 0,Y 433.872,Z 1066.131,A -85,B 0,C 180,E1 10309.151,E2 10309.151} C_VEL
LIN {X 0,Y 429.694,Z 1108.572,A -85,B 0,C 180,E1 10310.796,E2 10310.796} C_VEL
LIN {X 0,Y 424.538,Z 1148.3,A -85,B 0,C 180,E1 10313.197,E2 10313.197} C_VEL
LIN {X 0,Y 418.717,Z 1186.317,A -85,B 0,C 180,E1 10316.462,E2 10316.462} C_VEL
LIN {X 0,Y 413.263,Z 1220.474,A -85,B 0,C 180,E1 10320.47,E2 10320.47} C_VEL
LIN {X 0,Y 408.8,Z 1249.399,A -85,B 0,C 180,E1 10325.018,E2 10325.018} C_VEL
LIN {X 0,Y 405.561,Z 1273.659,A -85,B 0,C 180,E1 10330.156,E2 10330.156} C_VEL
LIN {X 0,Y 404.443,Z 1283.093,A -85,B 0,C 180,E1 10332.707,E2 10332.707} C_VEL
LIN {X 0,Y 399.851,Z 1289.868,A -85,B 0,C 180,E1 10334.92,E2 10334.92} C_VEL
LIN {X 0,Y 395.402,Z 1295.585,A -85,B 0,C 180,E1 10337.236,E2 10337.236} C_VEL
LIN {X 0,Y 394.967,Z 1305.071,A -85,B 0,C 180,E1 10342.319,E2 10342.319} C_VEL
LIN {X 0,Y 394.772,Z 1309.877,A -85,B 0,C 180,E1 10347.814,E2 10347.814} C_VEL
LIN {X 0,Y 394.818,Z 1309.796,A -85,B 0,C 180,E1 10352.195,E2 10352.195} C_VEL
LIN {X 0,Y 395.005,Z 1304.666,A -85,B 0,C 180,E1 10357.578,E2 10357.578} C_VEL
LIN {X 0,Y 395.563,Z 1294.587,A -85,B 0,C 180,E1 10362.676,E2 10362.676} C_VEL
LIN {X 0,Y 396.882,Z 1279.178,A -85,B 0,C 180,E1 10367.713,E2 10367.713} C_VEL
LIN {X 0,Y 399.162,Z 1258.001,A -85,B 0,C 180,E1 10372.591,E2 10372.591} C_VEL
LIN {X 0,Y 402.422,Z 1231.975,A -85,B 0,C 180,E1 10377.025,E2 10377.025} C_VEL
LIN {X 0,Y 406.657,Z 1199.783,A -85,B 0,C 180,E1 10381.15,E2 10381.15} C_VEL
LIN {X 0,Y 411.37,Z 1162.637,A -85,B 0,C 180,E1 10384.717,E2 10384.717} C_VEL
LIN {X 0,Y 416.386,Z 1121.137,A -85,B 0,C 180,E1 10387.65,E2 10387.65} C_VEL
LIN {X 0,Y 421.051,Z 1078.263,A -85,B 0,C 180,E1 10389.787,E2 10389.787} C_VEL
LIN {X 0,Y 421.76,Z 1064.366,A -85,B 0,C 180,E1 10390.38,E2 10390.38} C_VEL
LIN {X 0,Y 413.514,Z 1038.062,A -85,B 0,C 180,E1 10392.406,E2 10392.406} C_VEL
LIN {X 0,Y 408.118,Z 1015.812,A -85,B 0,C 180,E1 10394.13,E2 10394.13} C_VEL
LIN {X 0,Y 400.896,Z 1002.142,A -85,B 0,C 180,E1 10396.24,E2 10396.24} C_VEL
LIN {X 0,Y 396.715,Z 995.73,A -85,B 0,C 180,E1 10397.855,E2 10397.855} C_VEL
LIN {X 0,Y 393.054,Z 989.972,A -85,B 0,C 180,E1 10400.109,E2 10400.109} C_VEL
LIN {X 0,Y 392.938,Z 989.03,A -85,B 0,C 180,E1 10401.328,E2 10401.328} C_VEL
LIN {X 0,Y 393.134,Z 989.631,A -85,B 0,C 180,E1 10405.331,E2 10405.331} C_VEL
LIN {X 0,Y 397.568,Z 997.374,A -85,B 0,C 180,E1 10408.054,E2 10408.054} C_VEL
LIN {X 0,Y 403.552,Z 1008.914,A -85,B 0,C 180,E1 10410.254,E2 10410.254} C_VEL
LIN {X 0,Y 410.035,Z 1025.559,A -85,B 0,C 180,E1 10412.127,E2 10412.127} C_VEL
LIN {X 0,Y 412.171,Z 1037.086,A -85,B 0,C 180,E1 10412.889,E2 10412.889} C_VEL
LIN {X 0,Y 410.535,Z 1073.034,A -85,B 0,C 180,E1 10414.392,E2 10414.392} C_VEL
LIN {X 0,Y 408.17,Z 1101.246,A -85,B 0,C 180,E1 10416.439,E2 10416.439} C_VEL
LIN {X 0,Y 405.228,Z 1125.422,A -85,B 0,C 180,E1 10419.087,E2 10419.087} C_VEL
LIN {X 0,Y 402.079,Z 1146.862,A -85,B 0,C 180,E1 10422.528,E2 10422.528} C_VEL
LIN {X 0,Y 399.379,Z 1162.977,A -85,B 0,C 180,E1 10426.341,E2 10426.341} C_VEL
LIN {X 0,Y 397.529,Z 1174.707,A -85,B 0,C 180,E1 10430.771,E2 10430.771} C_VEL
LIN {X 0,Y 396.637,Z 1180.143,A -85,B 0,C 180,E1 10434.542,E2 10434.542} C_VEL
LIN {X 0,Y 396.331,Z 1181.735,A -85,B 0,C 180,E1 10437.818,E2 10437.818} C_VEL
LIN {X 0,Y 396.384,Z 1179.531,A -85,B 0,C 180,E1 10442.181,E2 10442.181} C_VEL
LIN {X 0,Y 396.725,Z 1172.276,A -85,B 0,C 180,E1 10446.552,E2 10446.552} C_VEL
LIN {X 0,Y 397.948,Z 1159.244,A -85,B 0,C 180,E1 10450.928,E2 10450.928} C_VEL
LIN {X 0,Y 400.02,Z 1140.246,A -85,B 0,C 180,E1 10455.03,E2 10455.03} C_VEL
LIN {X 0,Y 402.688,Z 1117.157,A -85,B 0,C 180,E1 10458.431,E2 10458.431} C_VEL
LIN {X 0,Y 405.393,Z 1090.079,A -85,B 0,C 180,E1 10461.182,E2 10461.182} C_VEL
LIN {X 0,Y 407.754,Z 1059.264,A -85,B 0,C 180,E1 10463.22,E2 10463.22} C_VEL
LIN {X 0,Y 408.269,Z 1030.989,A -85,B 0,C 180,E1 10464.359,E2 10464.359} C_VEL
LIN {X 0,Y 393.352,Z 989.03,A -85,B 0,C 180,E1 10466.578,E2 10466.578} C_VEL
LIN {X 0,Y 393.128,Z 989.03,A -85,B 0,C 180,E1 10472.504,E2 10472.504} C_VEL
LIN {X 0,Y 392.984,Z 989.03,A -85,B 0,C 180,E1 10479.819,E2 10479.819} C_VEL
LIN {X 0,Y 393.068,Z 989.03,A -85,B 0,C 180,E1 10486.834,E2 10486.834} C_VEL
LIN {X 0,Y 393.144,Z 989.567,A -85,B 0,C 180,E1 10488.327,E2 10488.327} C_VEL
LIN {X 0,Y 417.128,Z 1036.156,A -85,B 0,C 180,E1 10492.274,E2 10492.274} C_VEL
LIN {X 0,Y 423.648,Z 1053.172,A -85,B 0,C 180,E1 10493.512,E2 10493.512} C_VEL
LIN {X 0,Y 420.279,Z 1090.4,A -85,B 0,C 180,E1 10495.129,E2 10495.129} C_VEL
LIN {X 0,Y 415.852,Z 1124.597,A -85,B 0,C 180,E1 10497.48,E2 10497.48} C_VEL
LIN {X 0,Y 410.534,Z 1156.28,A -85,B 0,C 180,E1 10500.599,E2 10500.599} C_VEL
LIN {X 0,Y 405.372,Z 1183.615,A -85,B 0,C 180,E1 10504.353,E2 10504.353} C_VEL
LIN {X 0,Y 400.884,Z 1206.995,A -85,B 0,C 180,E1 10508.753,E2 10508.753} C_VEL
LIN {X 0,Y 397.715,Z 1225.023,A -85,B 0,C 180,E1 10513.462,E2 10513.462} C_VEL
LIN {X 0,Y 395.879,Z 1238.155,A -85,B 0,C 180,E1 10518.451,E2 10518.451} C_VEL
LIN {X 0,Y 395.102,Z 1246.226,A -85,B 0,C 180,E1 10523.416,E2 10523.416} C_VEL
LIN {X 0,Y 394.806,Z 1249.572,A -85,B 0,C 180,E1 10527.805,E2 10527.805} C_VEL
LIN {X 0,Y 394.921,Z 1249.525,A -85,B 0,C 180,E1 10532.186,E2 10532.186} C_VEL
LIN {X 0,Y 395.173,Z 1244.833,A -85,B 0,C 180,E1 10537.566,E2 10537.566} C_VEL
LIN {X 0,Y 396.198,Z 1235.468,A -85,B 0,C 180,E1 10542.646,E2 10542.646} C_VEL
LIN {X 0,Y 398.523,Z 1219.738,A -85,B 0,C 180,E1 10548.006,E2 10548.006} C_VEL
LIN {X 0,Y 402.268,Z 1199.406,A -85,B 0,C 180,E1 10552.744,E2 10552.744} C_VEL
LIN {X 0,Y 407.103,Z 1174.629,A -85,B 0,C 180,E1 10556.92,E2 10556.92} C_VEL
LIN {X 0,Y 412.635,Z 1144.231,A -85,B 0,C 180,E1 10560.62,E2 10560.62} C_VEL
LIN {X 0,Y 417.654,Z 1111.659,A -85,B 0,C 180,E1 10563.423,E2 10563.423} C_VEL
LIN {X 0,Y 421.771,Z 1076.832,A -85,B 0,C 180,E1 10565.461,E2 10565.461} C_VEL
LIN {X 0,Y 423.13,Z 1050.662,A -85,B 0,C 180,E1 10566.534,E2 10566.534} C_VEL
LIN {X 0,Y 407.471,Z 1016.593,A -85,B 0,C 180,E1 10569.17,E2 10569.17} C_VEL
LIN {X 0,Y 393.132,Z 990.348,A -85,B 0,C 180,E1 10571.552,E2 10571.552} C_VEL
LIN {X 0,Y 393.032,Z 989.03,A -85,B 0,C 180,E1 10571.686,E2 10571.686} C_VEL
LIN {X 0,Y 393.043,Z 989.03,A -85,B 0,C 180,E1 10576.837,E2 10576.837} C_VEL
LIN {X 0,Y 393.069,Z 989.03,A -85,B 0,C 180,E1 10583.721,E2 10583.721} C_VEL
LIN {X 0,Y 393.212,Z 989.03,A -85,B 0,C 180,E1 10590.075,E2 10590.075} C_VEL
LIN {X 0,Y 393.496,Z 989.03,A -85,B 0,C 180,E1 10597.452,E2 10597.452} C_VEL
LIN {X 0,Y 393.847,Z 989.03,A -85,B 0,C 180,E1 10604.444,E2 10604.444} C_VEL
LIN {X 0,Y 394.06,Z 989.03,A -85,B 0,C 180,E1 10611.19,E2 10611.19} C_VEL
LIN {X 0,Y 394.338,Z 989.03,A -85,B 0,C 180,E1 10617.807,E2 10617.807} C_VEL
LIN {X 0,Y 394.23,Z 989.03,A -85,B 0,C 180,E1 10624.391,E2 10624.391} C_VEL
LIN {X 0,Y 393.917,Z 989.03,A -85,B 0,C 180,E1 10631.043,E2 10631.043} C_VEL
LIN {X 0,Y 393.626,Z 989.03,A -85,B 0,C 180,E1 10637.859,E2 10637.859} C_VEL
LIN {X 0,Y 393.379,Z 989.03,A -85,B 0,C 180,E1 10644.958,E2 10644.958} C_VEL
LIN {X 0,Y 393.137,Z 989.03,A -85,B 0,C 180,E1 10652.504,E2 10652.504} C_VEL
LIN {X 0,Y 393.107,Z 989.03,A -85,B 0,C 180,E1 10659.854,E2 10659.854} C_VEL
LIN {X 0,Y 393.108,Z 989.338,A -85,B 0,C 180,E1 10661.549,E2 10661.549} C_VEL
LIN {X 0,Y 401.298,Z 1011.452,A -85,B 0,C 180,E1 10664.28,E2 10664.28} C_VEL
LIN {X 0,Y 422.957,Z 1059.708,A -85,B 0,C 180,E1 10667.918,E2 10667.918} C_VEL
LIN {X 0,Y 427.237,Z 1069.764,A -85,B 0,C 180,E1 10668.683,E2 10668.683} C_VEL
LIN {X 0,Y 422.495,Z 1111.854,A -85,B 0,C 180,E1 10670.412,E2 10670.412} C_VEL
LIN {X 0,Y 416.976,Z 1151.444,A -85,B 0,C 180,E1 10672.942,E2 10672.942} C_VEL
LIN {X 0,Y 411.102,Z 1188.05,A -85,B 0,C 180,E1 10676.218,E2 10676.218} C_VEL
LIN {X 0,Y 405.665,Z 1220.727,A -85,B 0,C 180,E1 10680.167,E2 10680.167} C_VEL
LIN {X 0,Y 401.084,Z 1249.324,A -85,B 0,C 180,E1 10684.79,E2 10684.79} C_VEL
LIN {X 0,Y 397.717,Z 1273.374,A -85,B 0,C 180,E1 10690.037,E2 10690.037} C_VEL
LIN {X 0,Y 395.767,Z 1291.673,A -85,B 0,C 180,E1 10695.654,E2 10695.654} C_VEL
LIN {X 0,Y 395.402,Z 1295.585,A -85,B 0,C 180,E1 10697.236,E2 10697.236} C_VEL
LIN {X 0,Y 392.586,Z 1299.295,A -85,B 0,C 180,E1 10699.03,E2 10699.03} C_VEL
LIN {X 0,Y 387.197,Z 1303.373,A -85,B 0,C 180,E1 10701.775,E2 10701.775} C_VEL
LIN {X 0,Y 387.112,Z 1303.814,A -85,B 0,C 180,E1 10702.094,E2 10702.094} C_VEL
LIN {X 0,Y 386.938,Z 1307.754,A -85,B 0,C 180,E1 10705.531,E2 10705.531} C_VEL
LIN {X 0,Y 386.962,Z 1309.684,A -85,B 0,C 180,E1 10710.004,E2 10710.004} C_VEL
LIN {X 0,Y 386.994,Z 1306.974,A -85,B 0,C 180,E1 10715.356,E2 10715.356} C_VEL
LIN {X 0,Y 387.331,Z 1298.906,A -85,B 0,C 180,E1 10720.669,E2 10720.669} C_VEL
LIN {X 0,Y 388.322,Z 1285.797,A -85,B 0,C 180,E1 10725.789,E2 10725.789} C_VEL
LIN {X 0,Y 390.269,Z 1267.117,A -85,B 0,C 180,E1 10730.823,E2 10730.823} C_VEL
LIN {X 0,Y 393.411,Z 1242.223,A -85,B 0,C 180,E1 10735.685,E2 10735.685} C_VEL
LIN {X 0,Y 397.141,Z 1213.862,A -85,B 0,C 180,E1 10739.763,E2 10739.763} C_VEL
LIN {X 0,Y 402.208,Z 1175.933,A -85,B 0,C 180,E1 10743.929,E2 10743.929} C_VEL
LIN {X 0,Y 407.594,Z 1134.612,A -85,B 0,C 180,E1 10747.283,E2 10747.283} C_VEL
LIN {X 0,Y 413.122,Z 1089,A -85,B 0,C 180,E1 10749.911,E2 10749.911} C_VEL
LIN {X 0,Y 415.209,Z 1067.462,A -85,B 0,C 180,E1 10750.864,E2 10750.864} C_VEL
LIN {X 0,Y 407.698,Z 1040.965,A -85,B 0,C 180,E1 10753.032,E2 10753.032} C_VEL
LIN {X 0,Y 403.076,Z 1019.697,A -85,B 0,C 180,E1 10754.815,E2 10754.815} C_VEL
LIN {X 0,Y 396.628,Z 1007.824,A -85,B 0,C 180,E1 10756.93,E2 10756.93} C_VEL
LIN {X 0,Y 393.31,Z 1002.461,A -85,B 0,C 180,E1 10758.389,E2 10758.389} C_VEL
LIN {X 0,Y 390.165,Z 996.398,A -85,B 0,C 180,E1 10760.847,E2 10760.847} C_VEL
LIN {X 0,Y 389.811,Z 996.234,A -85,B 0,C 180,E1 10764.504,E2 10764.504} C_VEL
LIN {X 0,Y 393.68,Z 1003.287,A -85,B 0,C 180,E1 10767.547,E2 10767.547} C_VEL
LIN {X 0,Y 399.434,Z 1015.601,A -85,B 0,C 180,E1 10769.975,E2 10769.975} C_VEL
LIN {X 0,Y 404.933,Z 1031.936,A -85,B 0,C 180,E1 10771.795,E2 10771.795} C_VEL
LIN {X 0,Y 405.8,Z 1039.697,A -85,B 0,C 180,E1 10772.285,E2 10772.285} C_VEL
LIN {X 0,Y 403.869,Z 1075.773,A -85,B 0,C 180,E1 10773.886,E2 10773.886} C_VEL
LIN {X 0,Y 401.291,Z 1103.875,A -85,B 0,C 180,E1 10776.01,E2 10776.01} C_VEL
LIN {X 0,Y 398.048,Z 1128.534,A -85,B 0,C 180,E1 10778.82,E2 10778.82} C_VEL
LIN {X 0,Y 394.789,Z 1148.806,A -85,B 0,C 180,E1 10782.195,E2 10782.195} C_VEL
LIN {X 0,Y 391.901,Z 1164.72,A -85,B 0,C 180,E1 10786.075,E2 10786.075} C_VEL
LIN {X 0,Y 389.889,Z 1176.316,A -85,B 0,C 180,E1 10790.588,E2 10790.588} C_VEL
LIN {X 0,Y 389.221,Z 1180.496,A -85,B 0,C 180,E1 10793.321,E2 10793.321} C_VEL
LIN {X 0,Y 388.586,Z 1183.168,A -85,B 0,C 180,E1 10797.774,E2 10797.774} C_VEL
LIN {X 0,Y 388.601,Z 1180.862,A -85,B 0,C 180,E1 10802.225,E2 10802.225} C_VEL
LIN {X 0,Y 388.966,Z 1173.502,A -85,B 0,C 180,E1 10806.683,E2 10806.683} C_VEL
LIN {X 0,Y 390.276,Z 1160.351,A -85,B 0,C 180,E1 10811.146,E2 10811.146} C_VEL
LIN {X 0,Y 392.437,Z 1141.22,A -85,B 0,C 180,E1 10815.328,E2 10815.328} C_VEL
LIN {X 0,Y 395.227,Z 1117.997,A -85,B 0,C 180,E1 10818.792,E2 10818.792} C_VEL
LIN {X 0,Y 398.143,Z 1089.942,A -85,B 0,C 180,E1 10821.661,E2 10821.661} C_VEL
LIN {X 0,Y 400.539,Z 1059.467,A -85,B 0,C 180,E1 10823.68,E2 10823.68} C_VEL
LIN {X 0,Y 401.152,Z 1033.151,A -85,B 0,C 180,E1 10824.758,E2 10824.758} C_VEL
LIN {X 0,Y 385.377,Z 989.03,A -85,B 0,C 180,E1 10827.131,E2 10827.131} C_VEL
LIN {X 0,Y 385.101,Z 989.03,A -85,B 0,C 180,E1 10833.268,E2 10833.268} C_VEL
LIN {X 0,Y 385.042,Z 989.03,A -85,B 0,C 180,E1 10838.83,E2 10838.83} C_VEL
LIN {X 0,Y 385.156,Z 989.03,A -85,B 0,C 180,E1 10846.265,E2 10846.265} C_VEL
LIN {X 0,Y 385.19,Z 989.03,A -85,B 0,C 180,E1 10847.2,E2 10847.2} C_VEL
LIN {X 0,Y 387.794,Z 994.848,A -85,B 0,C 180,E1 10847.74,E2 10847.74} C_VEL
LIN {X 0,Y 409.08,Z 1034.972,A -85,B 0,C 180,E1 10851.346,E2 10851.346} C_VEL
LIN {X 0,Y 417.165,Z 1056.02,A -85,B 0,C 180,E1 10852.951,E2 10852.951} C_VEL
LIN {X 0,Y 413.649,Z 1092.602,A -85,B 0,C 180,E1 10854.6,E2 10854.6} C_VEL
LIN {X 0,Y 408.968,Z 1126.817,A -85,B 0,C 180,E1 10857.021,E2 10857.021} C_VEL
LIN {X 0,Y 403.397,Z 1158.068,A -85,B 0,C 180,E1 10860.193,E2 10860.193} C_VEL
LIN {X 0,Y 397.87,Z 1185.899,A -85,B 0,C 180,E1 10864.135,E2 10864.135} C_VEL
LIN {X 0,Y 393.245,Z 1208.867,A -85,B 0,C 180,E1 10868.615,E2 10868.615} C_VEL
LIN {X 0,Y 389.811,Z 1227.322,A -85,B 0,C 180,E1 10873.696,E2 10873.696} C_VEL
LIN {X 0,Y 387.993,Z 1239.844,A -85,B 0,C 180,E1 10878.782,E2 10878.782} C_VEL
LIN {X 0,Y 387.139,Z 1248.064,A -85,B 0,C 180,E1 10884.494,E2 10884.494} C_VEL
LIN {X 0,Y 386.935,Z 1250.62,A -85,B 0,C 180,E1 10889.996,E2 10889.996} C_VEL
LIN {X 0,Y 387.16,Z 1247.983,A -85,B 0,C 180,E1 10895.489,E2 10895.489} C_VEL
LIN {X 0,Y 387.982,Z 1239.688,A -85,B 0,C 180,E1 10901.21,E2 10901.21} C_VEL
LIN {X 0,Y 389.891,Z 1227.076,A -85,B 0,C 180,E1 10906.292,E2 10906.292} C_VEL
LIN {X 0,Y 393.311,Z 1208.499,A -85,B 0,C 180,E1 10911.372,E2 10911.372} C_VEL
LIN {X 0,Y 397.933,Z 1185.419,A -85,B 0,C 180,E1 10915.851,E2 10915.851} C_VEL
LIN {X 0,Y 403.527,Z 1157.215,A -85,B 0,C 180,E1 10919.818,E2 10919.818} C_VEL
LIN {X 0,Y 409.035,Z 1125.906,A -85,B 0,C 180,E1 10922.963,E2 10922.963} C_VEL
LIN {X 0,Y 413.785,Z 1092.121,A -85,B 0,C 180,E1 10925.321,E2 10925.321} C_VEL
LIN {X 0,Y 417.159,Z 1055.812,A -85,B 0,C 180,E1 10926.961,E2 10926.961} C_VEL
LIN {X 0,Y 406.791,Z 1030.144,A -85,B 0,C 180,E1 10928.944,E2 10928.944} C_VEL
LIN {X 0,Y 386.585,Z 993.612,A -85,B 0,C 180,E1 10932.35,E2 10932.35} C_VEL
LIN {X 0,Y 385.111,Z 989.03,A -85,B 0,C 180,E1 10932.79,E2 10932.79} C_VEL
LIN {X 0,Y 385.068,Z 989.03,A -85,B 0,C 180,E1 10938.229,E2 10938.229} C_VEL
LIN {X 0,Y 385.158,Z 989.03,A -85,B 0,C 180,E1 10944.01,E2 10944.01} C_VEL
LIN {X 0,Y 385.343,Z 989.03,A -85,B 0,C 180,E1 10951.973,E2 10951.973} C_VEL
LIN {X 0,Y 385.756,Z 989.03,A -85,B 0,C 180,E1 10959.849,E2 10959.849} C_VEL
LIN {X 0,Y 386.011,Z 989.03,A -85,B 0,C 180,E1 10966.436,E2 10966.436} C_VEL
LIN {X 0,Y 386.293,Z 989.03,A -85,B 0,C 180,E1 10973.271,E2 10973.271} C_VEL
LIN {X 0,Y 386.569,Z 989.03,A -85,B 0,C 180,E1 10980,E2 10980} C_VEL
LIN {X 0,Y 386.29,Z 989.03,A -85,B 0,C 180,E1 10986.73,E2 10986.73} C_VEL
LIN {X 0,Y 385.909,Z 989.03,A -85,B 0,C 180,E1 10993.569,E2 10993.569} C_VEL
LIN {X 0,Y 385.586,Z 989.03,A -85,B 0,C 180,E1 11000.623,E2 11000.623} C_VEL
LIN {X 0,Y 385.334,Z 989.03,A -85,B 0,C 180,E1 11008.029,E2 11008.029} C_VEL
LIN {X 0,Y 385.156,Z 989.03,A -85,B 0,C 180,E1 11015.992,E2 11015.992} C_VEL
LIN {X 0,Y 385.172,Z 989.113,A -85,B 0,C 180,E1 11020.643,E2 11020.643} C_VEL
LIN {X 0,Y 392.866,Z 1010.052,A -85,B 0,C 180,E1 11023.289,E2 11023.289} C_VEL
LIN {X 0,Y 414.714,Z 1057.956,A -85,B 0,C 180,E1 11027.065,E2 11027.065} C_VEL
LIN {X 0,Y 420.352,Z 1073.271,A -85,B 0,C 180,E1 11028.198,E2 11028.198} C_VEL
LIN {X 0,Y 415.258,Z 1115.413,A -85,B 0,C 180,E1 11030.049,E2 11030.049} C_VEL
LIN {X 0,Y 409.388,Z 1154.582,A -85,B 0,C 180,E1 11032.684,E2 11032.684} C_VEL
LIN {X 0,Y 403.391,Z 1190.297,A -85,B 0,C 180,E1 11036.032,E2 11036.032} C_VEL
LIN {X 0,Y 397.772,Z 1222.864,A -85,B 0,C 180,E1 11040.142,E2 11040.142} C_VEL
LIN {X 0,Y 392.93,Z 1251.589,A -85,B 0,C 180,E1 11045.015,E2 11045.015} C_VEL
LIN {X 0,Y 389.716,Z 1274.176,A -85,B 0,C 180,E1 11050.2,E2 11050.2} C_VEL
LIN {X 0,Y 387.824,Z 1291.915,A -85,B 0,C 180,E1 11055.929,E2 11055.929} C_VEL
LIN {X 0,Y 387.153,Z 1302.29,A -85,B 0,C 180,E1 11061.035,E2 11061.035} C_VEL
LIN {X 0,Y 387.112,Z 1303.814,A -85,B 0,C 180,E1 11062.094,E2 11062.094} C_VEL
LIN {X 0,Y 384.518,Z 1306.127,A -85,B 0,C 180,E1 11063.976,E2 11063.976} C_VEL
LIN {X 0,Y 379.055,Z 1308.148,A -85,B 0,C 180,E1 11066.841,E2 11066.841} C_VEL
LIN {X 0,Y 378.978,Z 1308.224,A -85,B 0,C 180,E1 11067.173,E2 11067.173} C_VEL
LIN {X 0,Y 379.07,Z 1308.564,A -85,B 0,C 180,E1 11072.286,E2 11072.286} C_VEL
LIN {X 0,Y 379.223,Z 1304.839,A -85,B 0,C 180,E1 11076.861,E2 11076.861} C_VEL
LIN {X 0,Y 379.75,Z 1294.924,A -85,B 0,C 180,E1 11082.472,E2 11082.472} C_VEL
LIN {X 0,Y 381.107,Z 1280.155,A -85,B 0,C 180,E1 11087.684,E2 11087.684} C_VEL
LIN {X 0,Y 383.533,Z 1259.491,A -85,B 0,C 180,E1 11092.818,E2 11092.818} C_VEL
LIN {X 0,Y 387.177,Z 1233.253,A -85,B 0,C 180,E1 11097.571,E2 11097.571} C_VEL
LIN {X 0,Y 391.358,Z 1203.408,A -85,B 0,C 180,E1 11101.544,E2 11101.544} C_VEL
LIN {X 0,Y 397.17,Z 1159.166,A -85,B 0,C 180,E1 11105.853,E2 11105.853} C_VEL
LIN {X 0,Y 402.902,Z 1117.17,A -85,B 0,C 180,E1 11108.951,E2 11108.951} C_VEL
LIN {X 0,Y 408.741,Z 1072.717,A -85,B 0,C 180,E1 11111.257,E2 11111.257} C_VEL
LIN {X 0,Y 401.062,Z 1037.252,A -85,B 0,C 180,E1 11114.208,E2 11114.208} C_VEL
LIN {X 0,Y 397.723,Z 1022.956,A -85,B 0,C 180,E1 11115.661,E2 11115.661} C_VEL
LIN {X 0,Y 392.237,Z 1012.785,A -85,B 0,C 180,E1 11117.756,E2 11117.756} C_VEL
LIN {X 0,Y 389.537,Z 1008.636,A -85,B 0,C 180,E1 11119.139,E2 11119.139} C_VEL
LIN {X 0,Y 387.478,Z 1003.805,A -85,B 0,C 180,E1 11121.168,E2 11121.168} C_VEL
LIN {X 0,Y 387.04,Z 1003.601,A -85,B 0,C 180,E1 11124.211,E2 11124.211} C_VEL
LIN {X 0,Y 390.146,Z 1010.109,A -85,B 0,C 180,E1 11127.216,E2 11127.216} C_VEL
LIN {X 0,Y 395.189,Z 1021.901,A -85,B 0,C 180,E1 11129.633,E2 11129.633} C_VEL
LIN {X 0,Y 399.877,Z 1038.247,A -85,B 0,C 180,E1 11131.45,E2 11131.45} C_VEL
LIN {X 0,Y 397.246,Z 1079.517,A -85,B 0,C 180,E1 11133.417,E2 11133.417} C_VEL
LIN {X 0,Y 394.264,Z 1108.099,A -85,B 0,C 180,E1 11135.705,E2 11135.705} C_VEL
LIN {X 0,Y 390.738,Z 1132.375,A -85,B 0,C 180,E1 11138.653,E2 11138.653} C_VEL
LIN {X 0,Y 387.307,Z 1152.109,A -85,B 0,C 180,E1 11142.135,E2 11142.135} C_VEL
LIN {X 0,Y 384.139,Z 1168.287,A -85,B 0,C 180,E1 11146.367,E2 11146.367} C_VEL
LIN {X 0,Y 382.112,Z 1178.889,A -85,B 0,C 180,E1 11150.911,E2 11150.911} C_VEL
LIN {X 0,Y 381.129,Z 1183.942,A -85,B 0,C 180,E1 11155.458,E2 11155.458} C_VEL
LIN {X 0,Y 380.826,Z 1184.005,A -85,B 0,C 180,E1 11160,E2 11160} C_VEL
LIN {X 0,Y 380.984,Z 1179.104,A -85,B 0,C 180,E1 11164.543,E2 11164.543} C_VEL
LIN {X 0,Y 381.772,Z 1168.856,A -85,B 0,C 180,E1 11169.096,E2 11169.096} C_VEL
LIN {X 0,Y 383.579,Z 1153.364,A -85,B 0,C 180,E1 11173.362,E2 11173.362} C_VEL
LIN {X 0,Y 385.988,Z 1132.94,A -85,B 0,C 180,E1 11177.187,E2 11177.187} C_VEL
LIN {X 0,Y 389.064,Z 1107.863,A -85,B 0,C 180,E1 11180.429,E2 11180.429} C_VEL
LIN {X 0,Y 391.775,Z 1080.016,A -85,B 0,C 180,E1 11182.899,E2 11182.899} C_VEL
LIN {X 0,Y 394.014,Z 1048.078,A -85,B 0,C 180,E1 11184.673,E2 11184.673} C_VEL
LIN {X 0,Y 393.609,Z 1033.938,A -85,B 0,C 180,E1 11185.234,E2 11185.234} C_VEL
LIN {X 0,Y 377.417,Z 989.03,A -85,B 0,C 180,E1 11187.839,E2 11187.839} C_VEL
LIN {X 0,Y 377.148,Z 989.03,A -85,B 0,C 180,E1 11194.064,E2 11194.064} C_VEL
LIN {X 0,Y 377.018,Z 989.03,A -85,B 0,C 180,E1 11200.485,E2 11200.485} C_VEL
LIN {X 0,Y 377.268,Z 989.778,A -85,B 0,C 180,E1 11206.118,E2 11206.118} C_VEL
LIN {X 0,Y 401.33,Z 1034.464,A -85,B 0,C 180,E1 11210.424,E2 11210.424} C_VEL
LIN {X 0,Y 410.792,Z 1058.26,A -85,B 0,C 180,E1 11212.353,E2 11212.353} C_VEL
LIN {X 0,Y 407.063,Z 1094.454,A -85,B 0,C 180,E1 11214.029,E2 11214.029} C_VEL
LIN {X 0,Y 402.103,Z 1128.98,A -85,B 0,C 180,E1 11216.545,E2 11216.545} C_VEL
LIN {X 0,Y 396.223,Z 1160.244,A -85,B 0,C 180,E1 11219.823,E2 11219.823} C_VEL
LIN {X 0,Y 390.713,Z 1186.496,A -85,B 0,C 180,E1 11223.625,E2 11223.625} C_VEL
LIN {X 0,Y 385.814,Z 1209.47,A -85,B 0,C 180,E1 11228.182,E2 11228.182} C_VEL
LIN {X 0,Y 382.149,Z 1227.928,A -85,B 0,C 180,E1 11233.359,E2 11233.359} C_VEL
LIN {X 0,Y 380.186,Z 1240.45,A -85,B 0,C 180,E1 11238.548,E2 11238.548} C_VEL
LIN {X 0,Y 379.31,Z 1248.285,A -85,B 0,C 180,E1 11243.999,E2 11243.999} C_VEL
LIN {X 0,Y 379.058,Z 1251.221,A -85,B 0,C 180,E1 11249.996,E2 11249.996} C_VEL
LIN {X 0,Y 379.225,Z 1249.443,A -85,B 0,C 180,E1 11254.56,E2 11254.56} C_VEL
LIN {X 0,Y 379.908,Z 1242.449,A -85,B 0,C 180,E1 11260.292,E2 11260.292} C_VEL
LIN {X 0,Y 381.723,Z 1230.567,A -85,B 0,C 180,E1 11265.625,E2 11265.625} C_VEL
LIN {X 0,Y 385.113,Z 1212.647,A -85,B 0,C 180,E1 11270.946,E2 11270.946} C_VEL
LIN {X 0,Y 390.082,Z 1189.39,A -85,B 0,C 180,E1 11275.794,E2 11275.794} C_VEL
LIN {X 0,Y 395.929,Z 1161.295,A -85,B 0,C 180,E1 11279.956,E2 11279.956} C_VEL
LIN {X 0,Y 401.651,Z 1131.138,A -85,B 0,C 180,E1 11283.166,E2 11283.166} C_VEL
LIN {X 0,Y 406.73,Z 1097.557,A -85,B 0,C 180,E1 11285.688,E2 11285.688} C_VEL
LIN {X 0,Y 410.473,Z 1061.235,A -85,B 0,C 180,E1 11287.451,E2 11287.451} C_VEL
LIN {X 0,Y 410.08,Z 1054.764,A -85,B 0,C 180,E1 11287.784,E2 11287.784} C_VEL
LIN {X 0,Y 393.977,Z 1019.935,A -85,B 0,C 180,E1 11290.734,E2 11290.734} C_VEL
LIN {X 0,Y 377.33,Z 990.377,A -85,B 0,C 180,E1 11293.748,E2 11293.748} C_VEL
LIN {X 0,Y 377.193,Z 989.03,A -85,B 0,C 180,E1 11293.94,E2 11293.94} C_VEL
LIN {X 0,Y 377.134,Z 989.03,A -85,B 0,C 180,E1 11300.196,E2 11300.196} C_VEL
LIN {X 0,Y 377.193,Z 989.03,A -85,B 0,C 180,E1 11307.148,E2 11307.148} C_VEL
LIN {X 0,Y 377.449,Z 989.03,A -85,B 0,C 180,E1 11313.913,E2 11313.913} C_VEL
LIN {X 0,Y 377.818,Z 989.03,A -85,B 0,C 180,E1 11321.367,E2 11321.367} C_VEL
LIN {X 0,Y 378.161,Z 989.03,A -85,B 0,C 180,E1 11328.492,E2 11328.492} C_VEL
LIN {X 0,Y 378.462,Z 989.03,A -85,B 0,C 180,E1 11335.427,E2 11335.427} C_VEL
LIN {X 0,Y 378.645,Z 989.03,A -85,B 0,C 180,E1 11342.284,E2 11342.284} C_VEL
LIN {X 0,Y 378.164,Z 989.03,A -85,B 0,C 180,E1 11349.185,E2 11349.185} C_VEL
LIN {X 0,Y 377.795,Z 989.03,A -85,B 0,C 180,E1 11356.55,E2 11356.55} C_VEL
LIN {X 0,Y 377.533,Z 989.03,A -85,B 0,C 180,E1 11363.559,E2 11363.559} C_VEL
LIN {X 0,Y 377.35,Z 989.03,A -85,B 0,C 180,E1 11368.676,E2 11368.676} C_VEL
LIN {X 0,Y 377.196,Z 989.03,A -85,B 0,C 180,E1 11374.06,E2 11374.06} C_VEL
LIN {X 0,Y 377.323,Z 989.458,A -85,B 0,C 180,E1 11379.781,E2 11379.781} C_VEL
LIN {X 0,Y 384.571,Z 1008.982,A -85,B 0,C 180,E1 11382.292,E2 11382.292} C_VEL
LIN {X 0,Y 406.719,Z 1057.112,A -85,B 0,C 180,E1 11386.245,E2 11386.245} C_VEL
LIN {X 0,Y 413.503,Z 1076.019,A -85,B 0,C 180,E1 11387.681,E2 11387.681} C_VEL
LIN {X 0,Y 408.174,Z 1117.42,A -85,B 0,C 180,E1 11389.598,E2 11389.598} C_VEL
LIN {X 0,Y 401.884,Z 1157.147,A -85,B 0,C 180,E1 11392.379,E2 11392.379} C_VEL
LIN {X 0,Y 395.104,Z 1195.716,A -85,B 0,C 180,E1 11396.212,E2 11396.212} C_VEL
LIN {X 0,Y 389.342,Z 1227.639,A -85,B 0,C 180,E1 11400.544,E2 11400.544} C_VEL
LIN {X 0,Y 384.713,Z 1254.301,A -85,B 0,C 180,E1 11405.374,E2 11405.374} C_VEL
LIN {X 0,Y 381.602,Z 1275.918,A -85,B 0,C 180,E1 11410.664,E2 11410.664} C_VEL
LIN {X 0,Y 379.885,Z 1292.065,A -85,B 0,C 180,E1 11416.216,E2 11416.216} C_VEL
LIN {X 0,Y 379.231,Z 1303.257,A -85,B 0,C 180,E1 11421.999,E2 11421.999} C_VEL
LIN {X 0,Y 378.978,Z 1308.224,A -85,B 0,C 180,E1 11427.173,E2 11427.173} C_VEL
LIN {X 0,Y 376.601,Z 1308.893,A -85,B 0,C 180,E1 11429.125,E2 11429.125} C_VEL
LIN {X 0,Y 371.173,Z 1307.916,A -85,B 0,C 180,E1 11432.409,E2 11432.409} C_VEL
LIN {X 0,Y 371.326,Z 1304.233,A -85,B 0,C 180,E1 11437.007,E2 11437.007} C_VEL
LIN {X 0,Y 371.852,Z 1294.991,A -85,B 0,C 180,E1 11442.45,E2 11442.45} C_VEL
LIN {X 0,Y 373.299,Z 1279.945,A -85,B 0,C 180,E1 11447.944,E2 11447.944} C_VEL
LIN {X 0,Y 375.763,Z 1260.469,A -85,B 0,C 180,E1 11452.951,E2 11452.951} C_VEL
LIN {X 0,Y 379.615,Z 1234.495,A -85,B 0,C 180,E1 11457.85,E2 11457.85} C_VEL
LIN {X 0,Y 384.058,Z 1204.958,A -85,B 0,C 180,E1 11461.936,E2 11461.936} C_VEL
LIN {X 0,Y 388.309,Z 1172.455,A -85,B 0,C 180,E1 11465.242,E2 11465.242} C_VEL
LIN {X 0,Y 395.884,Z 1119.049,A -85,B 0,C 180,E1 11469.419,E2 11469.419} C_VEL
LIN {X 0,Y 402.029,Z 1076.258,A -85,B 0,C 180,E1 11471.794,E2 11471.794} C_VEL
LIN {X 0,Y 400.674,Z 1068.275,A -85,B 0,C 180,E1 11472.441,E2 11472.441} C_VEL
LIN {X 0,Y 393.728,Z 1029.17,A -85,B 0,C 180,E1 11476.07,E2 11476.07} C_VEL
LIN {X 0,Y 388.122,Z 1017.347,A -85,B 0,C 180,E1 11478.629,E2 11478.629} C_VEL
LIN {X 0,Y 385.034,Z 1011.317,A -85,B 0,C 180,E1 11481.168,E2 11481.168} C_VEL
LIN {X 0,Y 384.561,Z 1011.697,A -85,B 0,C 180,E1 11484.655,E2 11484.655} C_VEL
LIN {X 0,Y 387.249,Z 1018.721,A -85,B 0,C 180,E1 11487.341,E2 11487.341} C_VEL
LIN {X 0,Y 391.441,Z 1030.026,A -85,B 0,C 180,E1 11489.526,E2 11489.526} C_VEL
LIN {X 0,Y 393.969,Z 1042.665,A -85,B 0,C 180,E1 11490.848,E2 11490.848} C_VEL
LIN {X 0,Y 390.793,Z 1082.523,A -85,B 0,C 180,E1 11492.867,E2 11492.867} C_VEL
LIN {X 0,Y 387.472,Z 1111.048,A -85,B 0,C 180,E1 11495.251,E2 11495.251} C_VEL
LIN {X 0,Y 383.724,Z 1134.758,A -85,B 0,C 180,E1 11498.243,E2 11498.243} C_VEL
LIN {X 0,Y 379.883,Z 1155.004,A -85,B 0,C 180,E1 11501.969,E2 11501.969} C_VEL
LIN {X 0,Y 376.666,Z 1170.094,A -85,B 0,C 180,E1 11506.092,E2 11506.092} C_VEL
LIN {X 0,Y 374.472,Z 1180.537,A -85,B 0,C 180,E1 11510.724,E2 11510.724} C_VEL
LIN {X 0,Y 373.396,Z 1185.453,A -85,B 0,C 180,E1 11515.364,E2 11515.364} C_VEL
LIN {X 0,Y 373.05,Z 1185.391,A -85,B 0,C 180,E1 11520,E2 11520} C_VEL
LIN {X 0,Y 373.206,Z 1180.37,A -85,B 0,C 180,E1 11524.638,E2 11524.638} C_VEL
LIN {X 0,Y 374.065,Z 1169.986,A -85,B 0,C 180,E1 11529.285,E2 11529.285} C_VEL
LIN {X 0,Y 375.945,Z 1154.341,A -85,B 0,C 180,E1 11533.639,E2 11533.639} C_VEL
LIN {X 0,Y 378.542,Z 1133.31,A -85,B 0,C 180,E1 11537.604,E2 11537.604} C_VEL
LIN {X 0,Y 381.696,Z 1108.471,A -85,B 0,C 180,E1 11540.842,E2 11540.842} C_VEL
LIN {X 0,Y 384.568,Z 1079.672,A -85,B 0,C 180,E1 11543.408,E2 11543.408} C_VEL
LIN {X 0,Y 386.85,Z 1047.237,A -85,B 0,C 180,E1 11545.197,E2 11545.197} C_VEL
LIN {X 0,Y 386.273,Z 1035.329,A -85,B 0,C 180,E1 11545.688,E2 11545.688} C_VEL
LIN {X 0,Y 369.459,Z 989.03,A -85,B 0,C 180,E1 11548.432,E2 11548.432} C_VEL
LIN {X 0,Y 369.128,Z 989.03,A -85,B 0,C 180,E1 11555.144,E2 11555.144} C_VEL
LIN {X 0,Y 369.101,Z 989.03,A -85,B 0,C 180,E1 11562.608,E2 11562.608} C_VEL
LIN {X 0,Y 369.195,Z 989.729,A -85,B 0,C 180,E1 11564.883,E2 11564.883} C_VEL
LIN {X 0,Y 375.281,Z 1000.47,A -85,B 0,C 180,E1 11566.103,E2 11566.103} C_VEL
LIN {X 0,Y 395.95,Z 1038.883,A -85,B 0,C 180,E1 11569.897,E2 11569.897} C_VEL
LIN {X 0,Y 404.443,Z 1059.727,A -85,B 0,C 180,E1 11571.698,E2 11571.698} C_VEL
LIN {X 0,Y 400.547,Z 1096.463,A -85,B 0,C 180,E1 11573.454,E2 11573.454} C_VEL
LIN {X 0,Y 395.221,Z 1131.046,A -85,B 0,C 180,E1 11576.048,E2 11576.048} C_VEL
LIN {X 0,Y 389.347,Z 1160.956,A -85,B 0,C 180,E1 11579.251,E2 11579.251} C_VEL
LIN {X 0,Y 383.225,Z 1188.781,A -85,B 0,C 180,E1 11583.385,E2 11583.385} C_VEL
LIN {X 0,Y 377.868,Z 1212.427,A -85,B 0,C 180,E1 11588.316,E2 11588.316} C_VEL
LIN {X 0,Y 374.239,Z 1230.184,A -85,B 0,C 180,E1 11593.6,E2 11593.6} C_VEL
LIN {X 0,Y 372.142,Z 1243.179,A -85,B 0,C 180,E1 11599.481,E2 11599.481} C_VEL
LIN {X 0,Y 371.349,Z 1250.107,A -85,B 0,C 180,E1 11605.334,E2 11605.334} C_VEL
LIN {X 0,Y 371.181,Z 1251.822,A -85,B 0,C 180,E1 11609.996,E2 11609.996} C_VEL
LIN {X 0,Y 371.372,Z 1250.044,A -85,B 0,C 180,E1 11614.657,E2 11614.657} C_VEL
LIN {X 0,Y 372.13,Z 1243.053,A -85,B 0,C 180,E1 11620.51,E2 11620.51} C_VEL
LIN {X 0,Y 373.992,Z 1231.604,A -85,B 0,C 180,E1 11625.8,E2 11625.8} C_VEL
LIN {X 0,Y 377.411,Z 1214.408,A -85,B 0,C 180,E1 11631.087,E2 11631.087} C_VEL
LIN {X 0,Y 382.159,Z 1193.088,A -85,B 0,C 180,E1 11635.74,E2 11635.74} C_VEL
LIN {X 0,Y 388.289,Z 1165.93,A -85,B 0,C 180,E1 11640.02,E2 11640.02} C_VEL
LIN {X 0,Y 394.504,Z 1134.7,A -85,B 0,C 180,E1 11643.517,E2 11643.517} C_VEL
LIN {X 0,Y 399.869,Z 1101.303,A -85,B 0,C 180,E1 11646.143,E2 11646.143} C_VEL
LIN {X 0,Y 404.051,Z 1064.38,A -85,B 0,C 180,E1 11648.035,E2 11648.035} C_VEL
LIN {X 0,Y 403.955,Z 1058.111,A -85,B 0,C 180,E1 11648.332,E2 11648.332} C_VEL
LIN {X 0,Y 389.292,Z 1025.598,A -85,B 0,C 180,E1 11651.202,E2 11651.202} C_VEL
LIN {X 0,Y 370.84,Z 993.866,A -85,B 0,C 180,E1 11654.637,E2 11654.637} C_VEL
LIN {X 0,Y 369.164,Z 989.03,A -85,B 0,C 180,E1 11655.168,E2 11655.168} C_VEL
LIN {X 0,Y 369.166,Z 989.03,A -85,B 0,C 180,E1 11662.186,E2 11662.186} C_VEL
LIN {X 0,Y 369.306,Z 989.03,A -85,B 0,C 180,E1 11669.095,E2 11669.095} C_VEL
LIN {X 0,Y 369.6,Z 989.03,A -85,B 0,C 180,E1 11675.905,E2 11675.905} C_VEL
LIN {X 0,Y 369.993,Z 989.03,A -85,B 0,C 180,E1 11683.413,E2 11683.413} C_VEL
LIN {X 0,Y 370.273,Z 989.03,A -85,B 0,C 180,E1 11690.619,E2 11690.619} C_VEL
LIN {X 0,Y 370.637,Z 989.03,A -85,B 0,C 180,E1 11697.667,E2 11697.667} C_VEL
LIN {X 0,Y 370.742,Z 989.03,A -85,B 0,C 180,E1 11702.333,E2 11702.333} C_VEL
LIN {X 0,Y 370.232,Z 989.03,A -85,B 0,C 180,E1 11709.383,E2 11709.383} C_VEL
LIN {X 0,Y 369.895,Z 989.03,A -85,B 0,C 180,E1 11716.593,E2 11716.593} C_VEL
LIN {X 0,Y 369.548,Z 989.03,A -85,B 0,C 180,E1 11724.1,E2 11724.1} C_VEL
LIN {X 0,Y 369.297,Z 989.03,A -85,B 0,C 180,E1 11732.086,E2 11732.086} C_VEL
LIN {X 0,Y 369.359,Z 989.396,A -85,B 0,C 180,E1 11738.837,E2 11738.837} C_VEL
LIN {X 0,Y 376.073,Z 1007.457,A -85,B 0,C 180,E1 11741.222,E2 11741.222} C_VEL
LIN {X 0,Y 398.719,Z 1056.135,A -85,B 0,C 180,E1 11745.395,E2 11745.395} C_VEL
LIN {X 0,Y 406.667,Z 1078.442,A -85,B 0,C 180,E1 11747.157,E2 11747.157} C_VEL
LIN {X 0,Y 400.999,Z 1119.782,A -85,B 0,C 180,E1 11749.172,E2 11749.172} C_VEL
LIN {X 0,Y 394.308,Z 1159.63,A -85,B 0,C 180,E1 11752.091,E2 11752.091} C_VEL
LIN {X 0,Y 387.676,Z 1195.909,A -85,B 0,C 180,E1 11755.812,E2 11755.812} C_VEL
LIN {X 0,Y 381.671,Z 1227.926,A -85,B 0,C 180,E1 11760.273,E2 11760.273} C_VEL
LIN {X 0,Y 376.761,Z 1255.491,A -85,B 0,C 180,E1 11765.451,E2 11765.451} C_VEL
LIN {X 0,Y 373.442,Z 1277.52,A -85,B 0,C 180,E1 11771.144,E2 11771.144} C_VEL
LIN {X 0,Y 371.715,Z 1295.051,A -85,B 0,C 180,E1 11777.575,E2 11777.575} C_VEL
LIN {X 0,Y 371.264,Z 1304.237,A -85,B 0,C 180,E1 11783,E2 11783} C_VEL
LIN {X 0,Y 371.142,Z 1307.962,A -85,B 0,C 180,E1 11787.674,E2 11787.674} C_VEL
LIN {X 0,Y 371.173,Z 1307.916,A -85,B 0,C 180,E1 11792.409,E2 11792.409} C_VEL
LIN {X 0,Y 368.619,Z 1306.613,A -85,B 0,C 180,E1 11794.394,E2 11794.394} C_VEL
LIN {X 0,Y 363.437,Z 1302.9,A -85,B 0,C 180,E1 11797.707,E2 11797.707} C_VEL
LIN {X 0,Y 364.001,Z 1294.379,A -85,B 0,C 180,E1 11802.723,E2 11802.723} C_VEL
LIN {X 0,Y 365.509,Z 1279.511,A -85,B 0,C 180,E1 11808.282,E2 11808.282} C_VEL
LIN {X 0,Y 368.246,Z 1259.449,A -85,B 0,C 180,E1 11813.541,E2 11813.541} C_VEL
LIN {X 0,Y 372.348,Z 1233.878,A -85,B 0,C 180,E1 11818.443,E2 11818.443} C_VEL
LIN {X 0,Y 377.277,Z 1203.366,A -85,B 0,C 180,E1 11822.711,E2 11822.711} C_VEL
LIN {X 0,Y 381.875,Z 1170.636,A -85,B 0,C 180,E1 11826.052,E2 11826.052} C_VEL
LIN {X 0,Y 390.943,Z 1107.143,A -85,B 0,C 180,E1 11830.834,E2 11830.834} C_VEL
LIN {X 0,Y 395.671,Z 1075.396,A -85,B 0,C 180,E1 11832.612,E2 11832.612} C_VEL
LIN {X 0,Y 390.878,Z 1047.705,A -85,B 0,C 180,E1 11835.277,E2 11835.277} C_VEL
LIN {X 0,Y 388.929,Z 1033.519,A -85,B 0,C 180,E1 11836.81,E2 11836.81} C_VEL
LIN {X 0,Y 384.802,Z 1024.141,A -85,B 0,C 180,E1 11839.006,E2 11839.006} C_VEL
LIN {X 0,Y 382.472,Z 1020.048,A -85,B 0,C 180,E1 11840.858,E2 11840.858} C_VEL
LIN {X 0,Y 381.436,Z 1018.368,A -85,B 0,C 180,E1 11843.601,E2 11843.601} C_VEL
LIN {X 0,Y 382.502,Z 1022.271,A -85,B 0,C 180,E1 11845.952,E2 11845.952} C_VEL
LIN {X 0,Y 385.683,Z 1031.275,A -85,B 0,C 180,E1 11848.329,E2 11848.329} C_VEL
LIN {X 0,Y 388.485,Z 1043.534,A -85,B 0,C 180,E1 11849.996,E2 11849.996} C_VEL
LIN {X 0,Y 384.459,Z 1085.659,A -85,B 0,C 180,E1 11852.286,E2 11852.286} C_VEL
LIN {X 0,Y 380.769,Z 1114.146,A -85,B 0,C 180,E1 11854.785,E2 11854.785} C_VEL
LIN {X 0,Y 376.537,Z 1138.389,A -85,B 0,C 180,E1 11858.005,E2 11858.005} C_VEL
LIN {X 0,Y 372.501,Z 1157.943,A -85,B 0,C 180,E1 11861.795,E2 11861.795} C_VEL
LIN {X 0,Y 369.243,Z 1171.972,A -85,B 0,C 180,E1 11865.806,E2 11865.806} C_VEL
LIN {X 0,Y 366.846,Z 1182.212,A -85,B 0,C 180,E1 11870.53,E2 11870.53} C_VEL
LIN {X 0,Y 365.671,Z 1186.972,A -85,B 0,C 180,E1 11875.266,E2 11875.266} C_VEL
LIN {X 0,Y 365.292,Z 1186.773,A -85,B 0,C 180,E1 11880,E2 11880} C_VEL
LIN {X 0,Y 365.45,Z 1181.617,A -85,B 0,C 180,E1 11884.736,E2 11884.736} C_VEL
LIN {X 0,Y 366.348,Z 1171.079,A -85,B 0,C 180,E1 11889.483,E2 11889.483} C_VEL
LIN {X 0,Y 368.312,Z 1155.268,A -85,B 0,C 180,E1 11893.927,E2 11893.927} C_VEL
LIN {X 0,Y 370.883,Z 1135.385,A -85,B 0,C 180,E1 11897.766,E2 11897.766} C_VEL
LIN {X 0,Y 374.164,Z 1110.381,A -85,B 0,C 180,E1 11901.126,E2 11901.126} C_VEL
LIN {X 0,Y 377.26,Z 1080.959,A -85,B 0,C 180,E1 11903.815,E2 11903.815} C_VEL
LIN {X 0,Y 379.627,Z 1048.943,A -85,B 0,C 180,E1 11905.629,E2 11905.629} C_VEL
LIN {X 0,Y 379.13,Z 1037.464,A -85,B 0,C 180,E1 11906.122,E2 11906.122} C_VEL
LIN {X 0,Y 361.469,Z 989.03,A -85,B 0,C 180,E1 11909.147,E2 11909.147} C_VEL
LIN {X 0,Y 361.144,Z 989.03,A -85,B 0,C 180,E1 11915.799,E2 11915.799} C_VEL
LIN {X 0,Y 361.211,Z 989.03,A -85,B 0,C 180,E1 11923.539,E2 11923.539} C_VEL
LIN {X 0,Y 363.829,Z 994.853,A -85,B 0,C 180,E1 11924.16,E2 11924.16} C_VEL
LIN {X 0,Y 384.348,Z 1030.402,A -85,B 0,C 180,E1 11928.153,E2 11928.153} C_VEL
LIN {X 0,Y 398.058,Z 1062.137,A -85,B 0,C 180,E1 11931.056,E2 11931.056} C_VEL
LIN {X 0,Y 393.787,Z 1100.086,A -85,B 0,C 180,E1 11932.957,E2 11932.957} C_VEL
LIN {X 0,Y 388.074,Z 1134.6,A -85,B 0,C 180,E1 11935.673,E2 11935.673} C_VEL
LIN {X 0,Y 381.822,Z 1164.917,A -85,B 0,C 180,E1 11939.078,E2 11939.078} C_VEL
LIN {X 0,Y 375.358,Z 1192.581,A -85,B 0,C 180,E1 11943.43,E2 11943.43} C_VEL
LIN {X 0,Y 369.918,Z 1215.336,A -85,B 0,C 180,E1 11948.455,E2 11948.455} C_VEL
LIN {X 0,Y 366.291,Z 1232.438,A -85,B 0,C 180,E1 11953.849,E2 11953.849} C_VEL
LIN {X 0,Y 364.342,Z 1243.783,A -85,B 0,C 180,E1 11959.254,E2 11959.254} C_VEL
LIN {X 0,Y 363.5,Z 1250.708,A -85,B 0,C 180,E1 11965.233,E2 11965.233} C_VEL
LIN {X 0,Y 363.304,Z 1252.424,A -85,B 0,C 180,E1 11969.995,E2 11969.995} C_VEL
LIN {X 0,Y 363.525,Z 1250.483,A -85,B 0,C 180,E1 11974.999,E2 11974.999} C_VEL
LIN {X 0,Y 364.329,Z 1243.658,A -85,B 0,C 180,E1 11980.738,E2 11980.738} C_VEL
LIN {X 0,Y 366.326,Z 1232.212,A -85,B 0,C 180,E1 11986.14,E2 11986.14} C_VEL
LIN {X 0,Y 370.008,Z 1215.012,A -85,B 0,C 180,E1 11991.529,E2 11991.529} C_VEL
LIN {X 0,Y 375.017,Z 1193.691,A -85,B 0,C 180,E1 11996.267,E2 11996.267} C_VEL
LIN {X 0,Y 381.417,Z 1166.533,A -85,B 0,C 180,E1 12000.618,E2 12000.618} C_VEL
LIN {X 0,Y 387.928,Z 1135.291,A -85,B 0,C 180,E1 12004.163,E2 12004.163} C_VEL
LIN {X 0,Y 393.485,Z 1102.242,A -85,B 0,C 180,E1 12006.795,E2 12006.795} C_VEL
LIN {X 0,Y 397.903,Z 1064.844,A -85,B 0,C 180,E1 12008.735,E2 12008.735} C_VEL
LIN {X 0,Y 396.7,Z 1058.365,A -85,B 0,C 180,E1 12009.184,E2 12009.184} C_VEL
LIN {X 0,Y 382.377,Z 1026.882,A -85,B 0,C 180,E1 12012.098,E2 12012.098} C_VEL
LIN {X 0,Y 363.531,Z 994.59,A -85,B 0,C 180,E1 12015.784,E2 12015.784} C_VEL
LIN {X 0,Y 361.222,Z 989.03,A -85,B 0,C 180,E1 12016.44,E2 12016.44} C_VEL
LIN {X 0,Y 361.225,Z 989.03,A -85,B 0,C 180,E1 12022.529,E2 12022.529} C_VEL
LIN {X 0,Y 361.394,Z 989.03,A -85,B 0,C 180,E1 12029.932,E2 12029.932} C_VEL
LIN {X 0,Y 361.688,Z 989.03,A -85,B 0,C 180,E1 12036.609,E2 12036.609} C_VEL
LIN {X 0,Y 362.111,Z 989.03,A -85,B 0,C 180,E1 12043.419,E2 12043.419} C_VEL
LIN {X 0,Y 362.373,Z 989.03,A -85,B 0,C 180,E1 12050.412,E2 12050.412} C_VEL
LIN {X 0,Y 362.729,Z 989.03,A -85,B 0,C 180,E1 12057.616,E2 12057.616} C_VEL
LIN {X 0,Y 362.717,Z 989.03,A -85,B 0,C 180,E1 12063.221,E2 12063.221} C_VEL
LIN {X 0,Y 362.3,Z 989.03,A -85,B 0,C 180,E1 12069.59,E2 12069.59} C_VEL
LIN {X 0,Y 361.95,Z 989.03,A -85,B 0,C 180,E1 12076.968,E2 12076.968} C_VEL
LIN {X 0,Y 361.621,Z 989.03,A -85,B 0,C 180,E1 12084.663,E2 12084.663} C_VEL
LIN {X 0,Y 361.39,Z 989.03,A -85,B 0,C 180,E1 12090.07,E2 12090.07} C_VEL
LIN {X 0,Y 361.465,Z 989.694,A -85,B 0,C 180,E1 12097.91,E2 12097.91} C_VEL
LIN {X 0,Y 367.583,Z 1005.963,A -85,B 0,C 180,E1 12100.116,E2 12100.116} C_VEL
LIN {X 0,Y 390.988,Z 1055.909,A -85,B 0,C 180,E1 12104.581,E2 12104.581} C_VEL
LIN {X 0,Y 399.806,Z 1081.003,A -85,B 0,C 180,E1 12106.636,E2 12106.636} C_VEL
LIN {X 0,Y 393.642,Z 1123.065,A -85,B 0,C 180,E1 12108.796,E2 12108.796} C_VEL
LIN {X 0,Y 386.538,Z 1163.023,A -85,B 0,C 180,E1 12111.884,E2 12111.884} C_VEL
LIN {X 0,Y 379.828,Z 1198.404,A -85,B 0,C 180,E1 12115.695,E2 12115.695} C_VEL
LIN {X 0,Y 373.806,Z 1229.203,A -85,B 0,C 180,E1 12120.171,E2 12120.171} C_VEL
LIN {X 0,Y 368.929,Z 1255.58,A -85,B 0,C 180,E1 12125.308,E2 12125.308} C_VEL
LIN {X 0,Y 365.441,Z 1278.33,A -85,B 0,C 180,E1 12131.355,E2 12131.355} C_VEL
LIN {X 0,Y 364.039,Z 1292.767,A -85,B 0,C 180,E1 12136.572,E2 12136.572} C_VEL
LIN {X 0,Y 363.466,Z 1302.043,A -85,B 0,C 180,E1 12141.649,E2 12141.649} C_VEL
LIN {X 0,Y 363.288,Z 1306.112,A -85,B 0,C 180,E1 12145.46,E2 12145.46} C_VEL
LIN {X 0,Y 363.326,Z 1307.88,A -85,B 0,C 180,E1 12150.005,E2 12150.005} C_VEL
LIN {X 0,Y 363.384,Z 1304.893,A -85,B 0,C 180,E1 12155.964,E2 12155.964} C_VEL
LIN {X 0,Y 363.437,Z 1302.9,A -85,B 0,C 180,E1 12157.707,E2 12157.707} C_VEL
LIN {X 0,Y 361.089,Z 1300.016,A -85,B 0,C 180,E1 12159.7,E2 12159.7} C_VEL
LIN {X 0,Y 356.21,Z 1294.536,A -85,B 0,C 180,E1 12162.657,E2 12162.657} C_VEL
LIN {X 0,Y 356.155,Z 1293.802,A -85,B 0,C 180,E1 12162.992,E2 12162.992} C_VEL
LIN {X 0,Y 357.717,Z 1278.888,A -85,B 0,C 180,E1 12168.695,E2 12168.695} C_VEL
LIN {X 0,Y 360.775,Z 1258.658,A -85,B 0,C 180,E1 12174.1,E2 12174.1} C_VEL
LIN {X 0,Y 365.127,Z 1233.26,A -85,B 0,C 180,E1 12179.058,E2 12179.058} C_VEL
LIN {X 0,Y 370.389,Z 1202.757,A -85,B 0,C 180,E1 12183.398,E2 12183.398} C_VEL
LIN {X 0,Y 375.341,Z 1169.865,A -85,B 0,C 180,E1 12186.8,E2 12186.8} C_VEL
LIN {X 0,Y 386.146,Z 1098.044,A -85,B 0,C 180,E1 12192.109,E2 12192.109} C_VEL
LIN {X 0,Y 389.33,Z 1077.67,A -85,B 0,C 180,E1 12193.299,E2 12193.299} C_VEL
LIN {X 0,Y 385.724,Z 1050.241,A -85,B 0,C 180,E1 12196.092,E2 12196.092} C_VEL
LIN {X 0,Y 384.41,Z 1038.221,A -85,B 0,C 180,E1 12197.516,E2 12197.516} C_VEL
LIN {X 0,Y 381.107,Z 1030.542,A -85,B 0,C 180,E1 12199.574,E2 12199.574} C_VEL
LIN {X 0,Y 378.955,Z 1026.211,A -85,B 0,C 180,E1 12201.969,E2 12201.969} C_VEL
LIN {X 0,Y 378.65,Z 1025.752,A -85,B 0,C 180,E1 12203.29,E2 12203.29} C_VEL
LIN {X 0,Y 379.234,Z 1029.096,A -85,B 0,C 180,E1 12205.618,E2 12205.618} C_VEL
LIN {X 0,Y 381.49,Z 1036.871,A -85,B 0,C 180,E1 12207.788,E2 12207.788} C_VEL
LIN {X 0,Y 383.287,Z 1046.483,A -85,B 0,C 180,E1 12209.216,E2 12209.216} C_VEL
LIN {X 0,Y 378.13,Z 1089.879,A -85,B 0,C 180,E1 12211.746,E2 12211.746} C_VEL
LIN {X 0,Y 374.095,Z 1117.394,A -85,B 0,C 180,E1 12214.303,E2 12214.303} C_VEL
LIN {X 0,Y 369.598,Z 1140.939,A -85,B 0,C 180,E1 12217.569,E2 12217.569} C_VEL
LIN {X 0,Y 365.178,Z 1160.602,A -85,B 0,C 180,E1 12221.543,E2 12221.543} C_VEL
LIN {X 0,Y 361.428,Z 1175.429,A -85,B 0,C 180,E1 12226.11,E2 12226.11} C_VEL
LIN {X 0,Y 359.245,Z 1183.912,A -85,B 0,C 180,E1 12230.327,E2 12230.327} C_VEL
LIN {X 0,Y 357.952,Z 1188.504,A -85,B 0,C 180,E1 12235.163,E2 12235.163} C_VEL
LIN {X 0,Y 357.519,Z 1188.155,A -85,B 0,C 180,E1 12240,E2 12240} C_VEL
LIN {X 0,Y 357.671,Z 1182.86,A -85,B 0,C 180,E1 12244.84,E2 12244.84} C_VEL
LIN {X 0,Y 358.652,Z 1172.147,A -85,B 0,C 180,E1 12249.688,E2 12249.688} C_VEL
LIN {X 0,Y 360.687,Z 1156.155,A -85,B 0,C 180,E1 12254.228,E2 12254.228} C_VEL
LIN {X 0,Y 363.387,Z 1136.069,A -85,B 0,C 180,E1 12258.145,E2 12258.145} C_VEL
LIN {X 0,Y 366.827,Z 1110.825,A -85,B 0,C 180,E1 12261.57,E2 12261.57} C_VEL
LIN {X 0,Y 370.004,Z 1081.359,A -85,B 0,C 180,E1 12264.289,E2 12264.289} C_VEL
LIN {X 0,Y 372.456,Z 1049.219,A -85,B 0,C 180,E1 12266.13,E2 12266.13} C_VEL
LIN {X 0,Y 372.026,Z 1039.527,A -85,B 0,C 180,E1 12266.559,E2 12266.559} C_VEL
LIN {X 0,Y 353.514,Z 989.03,A -85,B 0,C 180,E1 12269.794,E2 12269.794} C_VEL
LIN {X 0,Y 353.21,Z 989.03,A -85,B 0,C 180,E1 12276.733,E2 12276.733} C_VEL
LIN {X 0,Y 353.293,Z 989.468,A -85,B 0,C 180,E1 12282.186,E2 12282.186} C_VEL
LIN {X 0,Y 355.972,Z 994.956,A -85,B 0,C 180,E1 12282.827,E2 12282.827} C_VEL
LIN {X 0,Y 374.935,Z 1026.896,A -85,B 0,C 180,E1 12286.743,E2 12286.743} C_VEL
LIN {X 0,Y 389.493,Z 1058.346,A -85,B 0,C 180,E1 12289.811,E2 12289.811} C_VEL
LIN {X 0,Y 391.74,Z 1066.446,A -85,B 0,C 180,E1 12290.486,E2 12290.486} C_VEL
LIN {X 0,Y 387.238,Z 1102.691,A -85,B 0,C 180,E1 12292.396,E2 12292.396} C_VEL
LIN {X 0,Y 381.278,Z 1136.665,A -85,B 0,C 180,E1 12295.145,E2 12295.145} C_VEL
LIN {X 0,Y 374.522,Z 1167.682,A -85,B 0,C 180,E1 12298.745,E2 12298.745} C_VEL
LIN {X 0,Y 367.84,Z 1194.709,A -85,B 0,C 180,E1 12303.17,E2 12303.17} C_VEL
LIN {X 0,Y 362.231,Z 1217.093,A -85,B 0,C 180,E1 12308.296,E2 12308.296} C_VEL
LIN {X 0,Y 358.32,Z 1234.511,A -85,B 0,C 180,E1 12314.108,E2 12314.108} C_VEL
LIN {X 0,Y 356.546,Z 1244.387,A -85,B 0,C 180,E1 12319.016,E2 12319.016} C_VEL
LIN {X 0,Y 355.646,Z 1251.308,A -85,B 0,C 180,E1 12325.127,E2 12325.127} C_VEL
LIN {X 0,Y 355.437,Z 1253.024,A -85,B 0,C 180,E1 12329.995,E2 12329.995} C_VEL
LIN {X 0,Y 355.695,Z 1250.298,A -85,B 0,C 180,E1 12336.084,E2 12336.084} C_VEL
LIN {X 0,Y 356.896,Z 1242.111,A -85,B 0,C 180,E1 12342.2,E2 12342.2} C_VEL
LIN {X 0,Y 359.376,Z 1229.509,A -85,B 0,C 180,E1 12347.719,E2 12347.719} C_VEL
LIN {X 0,Y 363.751,Z 1210.929,A -85,B 0,C 180,E1 12353.206,E2 12353.206} C_VEL
LIN {X 0,Y 369.38,Z 1188.391,A -85,B 0,C 180,E1 12357.908,E2 12357.908} C_VEL
LIN {X 0,Y 376.068,Z 1160.709,A -85,B 0,C 180,E1 12362.078,E2 12362.078} C_VEL
LIN {X 0,Y 382.88,Z 1128.261,A -85,B 0,C 180,E1 12365.54,E2 12365.54} C_VEL
LIN {X 0,Y 388.538,Z 1094.125,A -85,B 0,C 180,E1 12368.027,E2 12368.027} C_VEL
LIN {X 0,Y 391.494,Z 1063.789,A -85,B 0,C 180,E1 12369.569,E2 12369.569} C_VEL
LIN {X 0,Y 377.857,Z 1032.541,A -85,B 0,C 180,E1 12372.584,E2 12372.584} C_VEL
LIN {X 0,Y 358.989,Z 1000.005,A -85,B 0,C 180,E1 12376.39,E2 12376.39} C_VEL
LIN {X 0,Y 353.489,Z 990.652,A -85,B 0,C 180,E1 12377.627,E2 12377.627} C_VEL
LIN {X 0,Y 353.316,Z 989.03,A -85,B 0,C 180,E1 12377.858,E2 12377.858} C_VEL
LIN {X 0,Y 353.327,Z 989.03,A -85,B 0,C 180,E1 12384.233,E2 12384.233} C_VEL
LIN {X 0,Y 353.517,Z 989.03,A -85,B 0,C 180,E1 12391.997,E2 12391.997} C_VEL
LIN {X 0,Y 353.919,Z 989.03,A -85,B 0,C 180,E1 12400.058,E2 12400.058} C_VEL
LIN {X 0,Y 354.365,Z 989.03,A -85,B 0,C 180,E1 12407.708,E2 12407.708} C_VEL
LIN {X 0,Y 354.765,Z 989.03,A -85,B 0,C 180,E1 12415.121,E2 12415.121} C_VEL
LIN {X 0,Y 354.933,Z 989.03,A -85,B 0,C 180,E1 12422.437,E2 12422.437} C_VEL
LIN {X 0,Y 354.366,Z 989.03,A -85,B 0,C 180,E1 12429.807,E2 12429.807} C_VEL
LIN {X 0,Y 353.982,Z 989.03,A -85,B 0,C 180,E1 12437.362,E2 12437.362} C_VEL
LIN {X 0,Y 353.618,Z 989.03,A -85,B 0,C 180,E1 12445.26,E2 12445.26} C_VEL
LIN {X 0,Y 353.357,Z 989.03,A -85,B 0,C 180,E1 12451.346,E2 12451.346} C_VEL
LIN {X 0,Y 353.399,Z 989.466,A -85,B 0,C 180,E1 12456.876,E2 12456.876} C_VEL
LIN {X 0,Y 359.173,Z 1004.518,A -85,B 0,C 180,E1 12458.982,E2 12458.982} C_VEL
LIN {X 0,Y 383.317,Z 1055.82,A -85,B 0,C 180,E1 12463.759,E2 12463.759} C_VEL
LIN {X 0,Y 392.981,Z 1083.206,A -85,B 0,C 180,E1 12466.09,E2 12466.09} C_VEL
LIN {X 0,Y 386.613,Z 1124.219,A -85,B 0,C 180,E1 12468.289,E2 12468.289} C_VEL
LIN {X 0,Y 379.373,Z 1163.273,A -85,B 0,C 180,E1 12471.396,E2 12471.396} C_VEL
LIN {X 0,Y 372.215,Z 1199.545,A -85,B 0,C 180,E1 12475.423,E2 12475.423} C_VEL
LIN {X 0,Y 365.908,Z 1230.517,A -85,B 0,C 180,E1 12480.094,E2 12480.094} C_VEL
LIN {X 0,Y 360.797,Z 1257.429,A -85,B 0,C 180,E1 12485.582,E2 12485.582} C_VEL
LIN {X 0,Y 357.762,Z 1277.46,A -85,B 0,C 180,E1 12490.86,E2 12490.86} C_VEL
LIN {X 0,Y 356.193,Z 1292.243,A -85,B 0,C 180,E1 12496.311,E2 12496.311} C_VEL
LIN {X 0,Y 355.584,Z 1301.435,A -85,B 0,C 180,E1 12501.463,E2 12501.463} C_VEL
LIN {X 0,Y 355.412,Z 1305.341,A -85,B 0,C 180,E1 12505.133,E2 12505.133} C_VEL
LIN {X 0,Y 355.457,Z 1307.28,A -85,B 0,C 180,E1 12510.005,E2 12510.005} C_VEL
LIN {X 0,Y 355.432,Z 1305.338,A -85,B 0,C 180,E1 12514.876,E2 12514.876} C_VEL
LIN {X 0,Y 355.747,Z 1298.635,A -85,B 0,C 180,E1 12520.391,E2 12520.391} C_VEL
LIN {X 0,Y 356.155,Z 1293.802,A -85,B 0,C 180,E1 12522.992,E2 12522.992} C_VEL
LIN {X 0,Y 352.797,Z 1287.831,A -85,B 0,C 180,E1 12525.594,E2 12525.594} C_VEL
LIN {X 0,Y 349.716,Z 1281.021,A -85,B 0,C 180,E1 12528.2,E2 12528.2} C_VEL
LIN {X 0,Y 352.786,Z 1260.878,A -85,B 0,C 180,E1 12533.982,E2 12533.982} C_VEL
LIN {X 0,Y 357.261,Z 1236.228,A -85,B 0,C 180,E1 12539.067,E2 12539.067} C_VEL
LIN {X 0,Y 362.811,Z 1206.59,A -85,B 0,C 180,E1 12543.554,E2 12543.554} C_VEL
LIN {X 0,Y 368.191,Z 1173.602,A -85,B 0,C 180,E1 12547.172,E2 12547.172} C_VEL
LIN {X 0,Y 380.478,Z 1096.527,A -85,B 0,C 180,E1 12552.98,E2 12552.98} C_VEL
LIN {X 0,Y 383.112,Z 1079.777,A -85,B 0,C 180,E1 12554.044,E2 12554.044} C_VEL
LIN {X 0,Y 380.824,Z 1051.548,A -85,B 0,C 180,E1 12557.069,E2 12557.069} C_VEL
LIN {X 0,Y 380.371,Z 1044.167,A -85,B 0,C 180,E1 12558.009,E2 12558.009} C_VEL
LIN {X 0,Y 377.364,Z 1036.734,A -85,B 0,C 180,E1 12560.224,E2 12560.224} C_VEL
LIN {X 0,Y 375.797,Z 1033.137,A -85,B 0,C 180,E1 12562.965,E2 12562.965} C_VEL
LIN {X 0,Y 375.924,Z 1035.596,A -85,B 0,C 180,E1 12565.107,E2 12565.107} C_VEL
LIN {X 0,Y 377.51,Z 1043.115,A -85,B 0,C 180,E1 12567.348,E2 12567.348} C_VEL
LIN {X 0,Y 378.251,Z 1049.993,A -85,B 0,C 180,E1 12568.392,E2 12568.392} C_VEL
LIN {X 0,Y 372.063,Z 1093.407,A -85,B 0,C 180,E1 12571.121,E2 12571.121} C_VEL
LIN {X 0,Y 367.51,Z 1120.761,A -85,B 0,C 180,E1 12573.808,E2 12573.808} C_VEL
LIN {X 0,Y 362.509,Z 1144.552,A -85,B 0,C 180,E1 12577.275,E2 12577.275} C_VEL
LIN {X 0,Y 357.673,Z 1164.024,A -85,B 0,C 180,E1 12581.476,E2 12581.476} C_VEL
LIN {X 0,Y 354.013,Z 1177.365,A -85,B 0,C 180,E1 12585.813,E2 12585.813} C_VEL
LIN {X 0,Y 351.273,Z 1187.014,A -85,B 0,C 180,E1 12591.172,E2 12591.172} C_VEL
LIN {X 0,Y 350.229,Z 1190.046,A -85,B 0,C 180,E1 12595.056,E2 12595.056} C_VEL
LIN {X 0,Y 349.761,Z 1189.531,A -85,B 0,C 180,E1 12600,E2 12600} C_VEL
LIN {X 0,Y 349.919,Z 1184.074,A -85,B 0,C 180,E1 12604.947,E2 12604.947} C_VEL
LIN {X 0,Y 350.954,Z 1173.187,A -85,B 0,C 180,E1 12609.903,E2 12609.903} C_VEL
LIN {X 0,Y 353.089,Z 1157.033,A -85,B 0,C 180,E1 12614.54,E2 12614.54} C_VEL
LIN {X 0,Y 356.196,Z 1134.867,A -85,B 0,C 180,E1 12618.845,E2 12618.845} C_VEL
LIN {X 0,Y 359.652,Z 1109.941,A -85,B 0,C 180,E1 12622.185,E2 12622.185} C_VEL
LIN {X 0,Y 362.965,Z 1080.104,A -85,B 0,C 180,E1 12624.906,E2 12624.906} C_VEL
LIN {X 0,Y 365.363,Z 1047.539,A -85,B 0,C 180,E1 12626.723,E2 12626.723} C_VEL
LIN {X 0,Y 363.922,Z 1038.589,A -85,B 0,C 180,E1 12627.19,E2 12627.19} C_VEL
LIN {X 0,Y 345.519,Z 989.03,A -85,B 0,C 180,E1 12630.461,E2 12630.461} C_VEL
LIN {X 0,Y 345.181,Z 989.03,A -85,B 0,C 180,E1 12638.094,E2 12638.094} C_VEL
LIN {X 0,Y 345.357,Z 989.13,A -85,B 0,C 180,E1 12640.681,E2 12640.681} C_VEL
LIN {X 0,Y 347.669,Z 994.604,A -85,B 0,C 180,E1 12641.298,E2 12641.298} C_VEL
LIN {X 0,Y 366.901,Z 1026.014,A -85,B 0,C 180,E1 12645.51,E2 12645.51} C_VEL
LIN {X 0,Y 381.942,Z 1057.387,A -85,B 0,C 180,E1 12648.766,E2 12648.766} C_VEL
LIN {X 0,Y 385.536,Z 1068.676,A -85,B 0,C 180,E1 12649.815,E2 12649.815} C_VEL
LIN {X 0,Y 380.85,Z 1104.301,A -85,B 0,C 180,E1 12651.744,E2 12651.744} C_VEL
LIN {X 0,Y 374.828,Z 1137.244,A -85,B 0,C 180,E1 12654.456,E2 12654.456} C_VEL
LIN {X 0,Y 367.775,Z 1168.272,A -85,B 0,C 180,E1 12658.105,E2 12658.105} C_VEL
LIN {X 0,Y 360.738,Z 1195.308,A -85,B 0,C 180,E1 12662.598,E2 12662.598} C_VEL
LIN {X 0,Y 354.848,Z 1217.694,A -85,B 0,C 180,E1 12667.821,E2 12667.821} C_VEL
LIN {X 0,Y 350.657,Z 1235.116,A -85,B 0,C 180,E1 12673.751,E2 12673.751} C_VEL
LIN {X 0,Y 348.777,Z 1244.99,A -85,B 0,C 180,E1 12678.768,E2 12678.768} C_VEL
LIN {X 0,Y 347.795,Z 1251.909,A -85,B 0,C 180,E1 12685.017,E2 12685.017} C_VEL
LIN {X 0,Y 347.559,Z 1253.625,A -85,B 0,C 180,E1 12689.995,E2 12689.995} C_VEL
LIN {X 0,Y 347.845,Z 1250.901,A -85,B 0,C 180,E1 12696.222,E2 12696.222} C_VEL
LIN {X 0,Y 349.14,Z 1242.717,A -85,B 0,C 180,E1 12702.476,E2 12702.476} C_VEL
LIN {X 0,Y 352.096,Z 1228.613,A -85,B 0,C 180,E1 12708.669,E2 12708.669} C_VEL
LIN {X 0,Y 357.002,Z 1209.177,A -85,B 0,C 180,E1 12714.286,E2 12714.286} C_VEL
LIN {X 0,Y 363.353,Z 1185.361,A -85,B 0,C 180,E1 12719.142,E2 12719.142} C_VEL
LIN {X 0,Y 370.543,Z 1156.394,A -85,B 0,C 180,E1 12723.346,E2 12723.346} C_VEL
LIN {X 0,Y 377.13,Z 1125.551,A -85,B 0,C 180,E1 12726.522,E2 12726.522} C_VEL
LIN {X 0,Y 382.905,Z 1090.744,A -85,B 0,C 180,E1 12728.996,E2 12728.996} C_VEL
LIN {X 0,Y 385.189,Z 1066.283,A -85,B 0,C 180,E1 12730.254,E2 12730.254} C_VEL
LIN {X 0,Y 371.668,Z 1034.988,A -85,B 0,C 180,E1 12733.415,E2 12733.415} C_VEL
LIN {X 0,Y 352.057,Z 1001.091,A -85,B 0,C 180,E1 12737.573,E2 12737.573} C_VEL
LIN {X 0,Y 345.633,Z 990.831,A -85,B 0,C 180,E1 12739.092,E2 12739.092} C_VEL
LIN {X 0,Y 345.412,Z 989.03,A -85,B 0,C 180,E1 12739.443,E2 12739.443} C_VEL
LIN {X 0,Y 345.407,Z 989.03,A -85,B 0,C 180,E1 12746.1,E2 12746.1} C_VEL
LIN {X 0,Y 345.7,Z 989.03,A -85,B 0,C 180,E1 12754.121,E2 12754.121} C_VEL
LIN {X 0,Y 346.124,Z 989.03,A -85,B 0,C 180,E1 12762.232,E2 12762.232} C_VEL
LIN {X 0,Y 346.511,Z 989.03,A -85,B 0,C 180,E1 12769.969,E2 12769.969} C_VEL
LIN {X 0,Y 346.942,Z 989.03,A -85,B 0,C 180,E1 12777.508,E2 12777.508} C_VEL
LIN {X 0,Y 347.03,Z 989.03,A -85,B 0,C 180,E1 12782.493,E2 12782.493} C_VEL
LIN {X 0,Y 346.44,Z 989.03,A -85,B 0,C 180,E1 12790.034,E2 12790.034} C_VEL
LIN {X 0,Y 346.025,Z 989.03,A -85,B 0,C 180,E1 12797.774,E2 12797.774} C_VEL
LIN {X 0,Y 345.678,Z 989.03,A -85,B 0,C 180,E1 12805.882,E2 12805.882} C_VEL
LIN {X 0,Y 345.442,Z 989.03,A -85,B 0,C 180,E1 12813.909,E2 12813.909} C_VEL
LIN {X 0,Y 345.497,Z 989.468,A -85,B 0,C 180,E1 12815.857,E2 12815.857} C_VEL
LIN {X 0,Y 350.983,Z 1003.442,A -85,B 0,C 180,E1 12817.849,E2 12817.849} C_VEL
LIN {X 0,Y 375.525,Z 1055.541,A -85,B 0,C 180,E1 12822.89,E2 12822.89} C_VEL
LIN {X 0,Y 386.058,Z 1085.601,A -85,B 0,C 180,E1 12825.555,E2 12825.555} C_VEL
LIN {X 0,Y 379.23,Z 1127.344,A -85,B 0,C 180,E1 12827.919,E2 12827.919} C_VEL
LIN {X 0,Y 371.505,Z 1166.976,A -85,B 0,C 180,E1 12831.235,E2 12831.235} C_VEL
LIN {X 0,Y 364.248,Z 1202.039,A -85,B 0,C 180,E1 12835.329,E2 12835.329} C_VEL
LIN {X 0,Y 357.631,Z 1233.234,A -85,B 0,C 180,E1 12840.283,E2 12840.283} C_VEL
LIN {X 0,Y 352.563,Z 1260.887,A -85,B 0,C 180,E1 12846.012,E2 12846.012} C_VEL
LIN {X 0,Y 349.529,Z 1280.922,A -85,B 0,C 180,E1 12851.762,E2 12851.762} C_VEL
LIN {X 0,Y 348.062,Z 1294.676,A -85,B 0,C 180,E1 12857.485,E2 12857.485} C_VEL
LIN {X 0,Y 347.648,Z 1302.421,A -85,B 0,C 180,E1 12862.522,E2 12862.522} C_VEL
LIN {X 0,Y 347.532,Z 1306.158,A -85,B 0,C 180,E1 12867.516,E2 12867.516} C_VEL
LIN {X 0,Y 347.512,Z 1305.966,A -85,B 0,C 180,E1 12872.927,E2 12872.927} C_VEL
LIN {X 0,Y 347.716,Z 1300.817,A -85,B 0,C 180,E1 12878.742,E2 12878.742} C_VEL
LIN {X 0,Y 348.441,Z 1291.27,A -85,B 0,C 180,E1 12884.165,E2 12884.165} C_VEL
LIN {X 0,Y 349.716,Z 1281.021,A -85,B 0,C 180,E1 12888.2,E2 12888.2} C_VEL
LIN {X 0,Y 346.861,Z 1273.544,A -85,B 0,C 180,E1 12890.769,E2 12890.769} C_VEL
LIN {X 0,Y 344.435,Z 1265.073,A -85,B 0,C 180,E1 12893.291,E2 12893.291} C_VEL
LIN {X 0,Y 349.005,Z 1240.972,A -85,B 0,C 180,E1 12898.73,E2 12898.73} C_VEL
LIN {X 0,Y 354.931,Z 1211.348,A -85,B 0,C 180,E1 12903.559,E2 12903.559} C_VEL
LIN {X 0,Y 360.744,Z 1179.034,A -85,B 0,C 180,E1 12907.368,E2 12907.368} C_VEL
LIN {X 0,Y 365.774,Z 1143.595,A -85,B 0,C 180,E1 12910.34,E2 12910.34} C_VEL
LIN {X 0,Y 376.989,Z 1086.163,A -85,B 0,C 180,E1 12914.453,E2 12914.453} C_VEL
LIN {X 0,Y 376.274,Z 1074.798,A -85,B 0,C 180,E1 12915.697,E2 12915.697} C_VEL
LIN {X 0,Y 376.334,Z 1050.181,A -85,B 0,C 180,E1 12918.483,E2 12918.483} C_VEL
LIN {X 0,Y 373.843,Z 1043.168,A -85,B 0,C 180,E1 12920.745,E2 12920.745} C_VEL
LIN {X 0,Y 372.845,Z 1040.813,A -85,B 0,C 180,E1 12922.622,E2 12922.622} C_VEL
LIN {X 0,Y 372.717,Z 1042.443,A -85,B 0,C 180,E1 12924.762,E2 12924.762} C_VEL
LIN {X 0,Y 373.629,Z 1049.769,A -85,B 0,C 180,E1 12926.966,E2 12926.966} C_VEL
LIN {X 0,Y 373.573,Z 1053.781,A -85,B 0,C 180,E1 12927.532,E2 12927.532} C_VEL
LIN {X 0,Y 366.058,Z 1097.691,A -85,B 0,C 180,E1 12930.522,E2 12930.522} C_VEL
LIN {X 0,Y 361.011,Z 1124.323,A -85,B 0,C 180,E1 12933.299,E2 12933.299} C_VEL
LIN {X 0,Y 355.666,Z 1147.334,A -85,B 0,C 180,E1 12936.813,E2 12936.813} C_VEL
LIN {X 0,Y 350.492,Z 1166.371,A -85,B 0,C 180,E1 12941.106,E2 12941.106} C_VEL
LIN {X 0,Y 346.609,Z 1179.333,A -85,B 0,C 180,E1 12945.503,E2 12945.503} C_VEL
LIN {X 0,Y 343.657,Z 1188.725,A -85,B 0,C 180,E1 12950.975,E2 12950.975} C_VEL
LIN {X 0,Y 342.505,Z 1191.604,A -85,B 0,C 180,E1 12954.945,E2 12954.945} C_VEL
LIN {X 0,Y 341.98,Z 1190.906,A -85,B 0,C 180,E1 12960,E2 12960} C_VEL
LIN {X 0,Y 342.145,Z 1185.278,A -85,B 0,C 180,E1 12965.06,E2 12965.06} C_VEL
LIN {X 0,Y 343.26,Z 1174.2,A -85,B 0,C 180,E1 12970.127,E2 12970.127} C_VEL
LIN {X 0,Y 345.473,Z 1157.834,A -85,B 0,C 180,E1 12974.868,E2 12974.868} C_VEL
LIN {X 0,Y 348.447,Z 1137.334,A -85,B 0,C 180,E1 12978.952,E2 12978.952} C_VEL
LIN {X 0,Y 352.163,Z 1111.615,A -85,B 0,C 180,E1 12982.516,E2 12982.516} C_VEL
LIN {X 0,Y 355.598,Z 1081.862,A -85,B 0,C 180,E1 12985.313,E2 12985.313} C_VEL
LIN {X 0,Y 358.173,Z 1049.674,A -85,B 0,C 180,E1 12987.177,E2 12987.177} C_VEL
LIN {X 0,Y 356.807,Z 1040.683,A -85,B 0,C 180,E1 12987.662,E2 12987.662} C_VEL
LIN {X 0,Y 337.553,Z 989.03,A -85,B 0,C 180,E1 12991.257,E2 12991.257} C_VEL
LIN {X 0,Y 337.33,Z 989.366,A -85,B 0,C 180,E1 12999.053,E2 12999.053} C_VEL
LIN {X 0,Y 339.846,Z 994.779,A -85,B 0,C 180,E1 12999.758,E2 12999.758} C_VEL
LIN {X 0,Y 357.97,Z 1023.445,A -85,B 0,C 180,E1 13003.995,E2 13003.995} C_VEL
LIN {X 0,Y 373.876,Z 1055.175,A -85,B 0,C 180,E1 13007.545,E2 13007.545} C_VEL
LIN {X 0,Y 379.313,Z 1071.473,A -85,B 0,C 180,E1 13009.152,E2 13009.152} C_VEL
LIN {X 0,Y 374.371,Z 1106.917,A -85,B 0,C 180,E1 13011.142,E2 13011.142} C_VEL
LIN {X 0,Y 367.726,Z 1141.047,A -85,B 0,C 180,E1 13014.057,E2 13014.057} C_VEL
LIN {X 0,Y 360.198,Z 1171.912,A -85,B 0,C 180,E1 13017.885,E2 13017.885} C_VEL
LIN {X 0,Y 353.249,Z 1197.448,A -85,B 0,C 180,E1 13022.312,E2 13022.312} C_VEL
LIN {X 0,Y 347.187,Z 1219.406,A -85,B 0,C 180,E1 13027.641,E2 13027.641} C_VEL
LIN {X 0,Y 343.004,Z 1235.722,A -85,B 0,C 180,E1 13033.378,E2 13033.378} C_VEL
LIN {X 0,Y 341.009,Z 1245.593,A -85,B 0,C 180,E1 13038.509,E2 13038.509} C_VEL
LIN {X 0,Y 339.947,Z 1252.51,A -85,B 0,C 180,E1 13044.902,E2 13044.902} C_VEL
LIN {X 0,Y 339.692,Z 1254.226,A -85,B 0,C 180,E1 13049.995,E2 13049.995} C_VEL
LIN {X 0,Y 339.992,Z 1251.504,A -85,B 0,C 180,E1 13056.366,E2 13056.366} C_VEL
LIN {X 0,Y 341.406,Z 1243.322,A -85,B 0,C 180,E1 13062.763,E2 13062.763} C_VEL
LIN {X 0,Y 344.455,Z 1229.645,A -85,B 0,C 180,E1 13068.945,E2 13068.945} C_VEL
LIN {X 0,Y 349.367,Z 1211.171,A -85,B 0,C 180,E1 13074.481,E2 13074.481} C_VEL
LIN {X 0,Y 355.724,Z 1188.423,A -85,B 0,C 180,E1 13079.321,E2 13079.321} C_VEL
LIN {X 0,Y 363.196,Z 1160.195,A -85,B 0,C 180,E1 13083.633,E2 13083.633} C_VEL
LIN {X 0,Y 370.433,Z 1127.92,A -85,B 0,C 180,E1 13087.095,E2 13087.095} C_VEL
LIN {X 0,Y 376.47,Z 1093.659,A -85,B 0,C 180,E1 13089.607,E2 13089.607} C_VEL
LIN {X 0,Y 378.977,Z 1068.77,A -85,B 0,C 180,E1 13090.953,E2 13090.953} C_VEL
LIN {X 0,Y 365.416,Z 1037.256,A -85,B 0,C 180,E1 13094.295,E2 13094.295} C_VEL
LIN {X 0,Y 347.269,Z 1006.086,A -85,B 0,C 180,E1 13098.304,E2 13098.304} C_VEL
LIN {X 0,Y 339.077,Z 993.81,A -85,B 0,C 180,E1 13100.309,E2 13100.309} C_VEL
LIN {X 0,Y 337.435,Z 989.03,A -85,B 0,C 180,E1 13100.824,E2 13100.824} C_VEL
LIN {X 0,Y 337.52,Z 989.03,A -85,B 0,C 180,E1 13108.147,E2 13108.147} C_VEL
LIN {X 0,Y 337.868,Z 989.03,A -85,B 0,C 180,E1 13116.301,E2 13116.301} C_VEL
LIN {X 0,Y 338.145,Z 989.03,A -85,B 0,C 180,E1 13121.799,E2 13121.799} C_VEL
LIN {X 0,Y 338.571,Z 989.03,A -85,B 0,C 180,E1 13129.731,E2 13129.731} C_VEL
LIN {X 0,Y 339.031,Z 989.03,A -85,B 0,C 180,E1 13137.45,E2 13137.45} C_VEL
LIN {X 0,Y 339.113,Z 989.03,A -85,B 0,C 180,E1 13142.551,E2 13142.551} C_VEL
LIN {X 0,Y 338.501,Z 989.03,A -85,B 0,C 180,E1 13150.272,E2 13150.272} C_VEL
LIN {X 0,Y 338.05,Z 989.03,A -85,B 0,C 180,E1 13158.208,E2 13158.208} C_VEL
LIN {X 0,Y 337.827,Z 989.03,A -85,B 0,C 180,E1 13163.703,E2 13163.703} C_VEL
LIN {X 0,Y 337.521,Z 989.03,A -85,B 0,C 180,E1 13171.853,E2 13171.853} C_VEL
LIN {X 0,Y 337.555,Z 989.582,A -85,B 0,C 180,E1 13174.814,E2 13174.814} C_VEL
LIN {X 0,Y 342.645,Z 1002.221,A -85,B 0,C 180,E1 13176.647,E2 13176.647} C_VEL
LIN {X 0,Y 367.505,Z 1054.871,A -85,B 0,C 180,E1 13181.951,E2 13181.951} C_VEL
LIN {X 0,Y 379.312,Z 1086.611,A -85,B 0,C 180,E1 13184.949,E2 13184.949} C_VEL
LIN {X 0,Y 372.307,Z 1127.694,A -85,B 0,C 180,E1 13187.346,E2 13187.346} C_VEL
LIN {X 0,Y 364.274,Z 1167.212,A -85,B 0,C 180,E1 13190.74,E2 13190.74} C_VEL
LIN {X 0,Y 356.786,Z 1202.069,A -85,B 0,C 180,E1 13194.917,E2 13194.917} C_VEL
LIN {X 0,Y 348.718,Z 1241.099,A -85,B 0,C 180,E1 13201.282,E2 13201.282} C_VEL
LIN {X 0,Y 344.109,Z 1265.3,A -85,B 0,C 180,E1 13206.759,E2 13206.759} C_VEL
LIN {X 0,Y 341.286,Z 1283.908,A -85,B 0,C 180,E1 13212.64,E2 13212.64} C_VEL
LIN {X 0,Y 340.101,Z 1296.571,A -85,B 0,C 180,E1 13218.581,E2 13218.581} C_VEL
LIN {X 0,Y 339.665,Z 1303.08,A -85,B 0,C 180,E1 13223.628,E2 13223.628} C_VEL
LIN {X 0,Y 339.645,Z 1305.556,A -85,B 0,C 180,E1 13227.458,E2 13227.458} C_VEL
LIN {X 0,Y 339.677,Z 1305.555,A -85,B 0,C 180,E1 13232.551,E2 13232.551} C_VEL
LIN {X 0,Y 339.785,Z 1301.809,A -85,B 0,C 180,E1 13237.662,E2 13237.662} C_VEL
LIN {X 0,Y 340.411,Z 1292.85,A -85,B 0,C 180,E1 13243.463,E2 13243.463} C_VEL
LIN {X 0,Y 342.119,Z 1278.641,A -85,B 0,C 180,E1 13249.251,E2 13249.251} C_VEL
LIN {X 0,Y 344.435,Z 1265.073,A -85,B 0,C 180,E1 13253.291,E2 13253.291} C_VEL
LIN {X 0,Y 342.263,Z 1256.081,A -85,B 0,C 180,E1 13255.785,E2 13255.785} C_VEL
LIN {X 0,Y 340.332,Z 1247.6,A -85,B 0,C 180,E1 13257.92,E2 13257.92} C_VEL
LIN {X 0,Y 340.556,Z 1246.238,A -85,B 0,C 180,E1 13258.207,E2 13258.207} C_VEL
LIN {X 0,Y 346.502,Z 1218.446,A -85,B 0,C 180,E1 13263.175,E2 13263.175} C_VEL
LIN {X 0,Y 352.716,Z 1187.06,A -85,B 0,C 180,E1 13267.266,E2 13267.266} C_VEL
LIN {X 0,Y 358.507,Z 1151.814,A -85,B 0,C 180,E1 13270.521,E2 13270.521} C_VEL
LIN {X 0,Y 362.78,Z 1125.016,A -85,B 0,C 180,E1 13272.539,E2 13272.539} C_VEL
LIN {X 0,Y 371.636,Z 1085.749,A -85,B 0,C 180,E1 13275.454,E2 13275.454} C_VEL
LIN {X 0,Y 371.843,Z 1059.251,A -85,B 0,C 180,E1 13278.664,E2 13278.664} C_VEL
LIN {X 0,Y 371.803,Z 1054.168,A -85,B 0,C 180,E1 13279.507,E2 13279.507} C_VEL
LIN {X 0,Y 370.314,Z 1049.494,A -85,B 0,C 180,E1 13281.347,E2 13281.347} C_VEL
LIN {X 0,Y 369.866,Z 1048.483,A -85,B 0,C 180,E1 13282.269,E2 13282.269} C_VEL
LIN {X 0,Y 369.627,Z 1050.818,A -85,B 0,C 180,E1 13285.143,E2 13285.143} C_VEL
LIN {X 0,Y 369.46,Z 1057.287,A -85,B 0,C 180,E1 13286.599,E2 13286.599} C_VEL
LIN {X 0,Y 360.904,Z 1098.435,A -85,B 0,C 180,E1 13289.56,E2 13289.56} C_VEL
LIN {X 0,Y 354.858,Z 1126.947,A -85,B 0,C 180,E1 13292.628,E2 13292.628} C_VEL
LIN {X 0,Y 348.777,Z 1150.573,A -85,B 0,C 180,E1 13296.409,E2 13296.409} C_VEL
LIN {X 0,Y 343.359,Z 1168.769,A -85,B 0,C 180,E1 13300.712,E2 13300.712} C_VEL
LIN {X 0,Y 338.819,Z 1182.759,A -85,B 0,C 180,E1 13305.821,E2 13305.821} C_VEL
LIN {X 0,Y 335.791,Z 1191.059,A -85,B 0,C 180,E1 13311.406,E2 13311.406} C_VEL
LIN {X 0,Y 334.812,Z 1193.163,A -85,B 0,C 180,E1 13314.828,E2 13314.828} C_VEL
LIN {X 0,Y 334.221,Z 1192.281,A -85,B 0,C 180,E1 13319.999,E2 13319.999} C_VEL
LIN {X 0,Y 334.369,Z 1186.461,A -85,B 0,C 180,E1 13325.178,E2 13325.178} C_VEL
LIN {X 0,Y 335.554,Z 1175.207,A -85,B 0,C 180,E1 13330.362,E2 13330.362} C_VEL
LIN {X 0,Y 337.883,Z 1158.638,A -85,B 0,C 180,E1 13335.21,E2 13335.21} C_VEL
LIN {X 0,Y 341.004,Z 1137.896,A -85,B 0,C 180,E1 13339.382,E2 13339.382} C_VEL
LIN {X 0,Y 344.913,Z 1111.497,A -85,B 0,C 180,E1 13343.066,E2 13343.066} C_VEL
LIN {X 0,Y 348.443,Z 1081.632,A -85,B 0,C 180,E1 13345.871,E2 13345.871} C_VEL
LIN {X 0,Y 351.029,Z 1049.493,A -85,B 0,C 180,E1 13347.735,E2 13347.735} C_VEL
LIN {X 0,Y 342.057,Z 1021.593,A -85,B 0,C 180,E1 13349.544,E2 13349.544} C_VEL
LIN {X 0,Y 329.611,Z 989.03,A -85,B 0,C 180,E1 13351.996,E2 13351.996} C_VEL
LIN {X 0,Y 329.29,Z 989.076,A -85,B 0,C 180,E1 13357.26,E2 13357.26} C_VEL
LIN {X 0,Y 331.454,Z 994.437,A -85,B 0,C 180,E1 13357.943,E2 13357.943} C_VEL
LIN {X 0,Y 338.352,Z 1004.291,A -85,B 0,C 180,E1 13359.762,E2 13359.762} C_VEL
LIN {X 0,Y 356.813,Z 1034.833,A -85,B 0,C 180,E1 13364.127,E2 13364.127} C_VEL
LIN {X 0,Y 370.556,Z 1065.009,A -85,B 0,C 180,E1 13367.554,E2 13367.554} C_VEL
LIN {X 0,Y 373.112,Z 1074.47,A -85,B 0,C 180,E1 13368.474,E2 13368.474} C_VEL
LIN {X 0,Y 367.736,Z 1110.581,A -85,B 0,C 180,E1 13370.59,E2 13370.59} C_VEL
LIN {X 0,Y 360.702,Z 1144.281,A -85,B 0,C 180,E1 13373.609,E2 13373.609} C_VEL
LIN {X 0,Y 352.917,Z 1174.537,A -85,B 0,C 180,E1 13377.503,E2 13377.503} C_VEL
LIN {X 0,Y 345.342,Z 1201.057,A -85,B 0,C 180,E1 13382.331,E2 13382.331} C_VEL
LIN {X 0,Y 339.197,Z 1222.088,A -85,B 0,C 180,E1 13387.775,E2 13387.775} C_VEL
LIN {X 0,Y 335.028,Z 1237.785,A -85,B 0,C 180,E1 13393.644,E2 13393.644} C_VEL
LIN {X 0,Y 332.868,Z 1248.02,A -85,B 0,C 180,E1 13399.547,E2 13399.547} C_VEL
LIN {X 0,Y 332.074,Z 1253.113,A -85,B 0,C 180,E1 13404.78,E2 13404.78} C_VEL
LIN {X 0,Y 331.829,Z 1254.826,A -85,B 0,C 180,E1 13409.995,E2 13409.995} C_VEL
LIN {X 0,Y 332.169,Z 1252.105,A -85,B 0,C 180,E1 13416.516,E2 13416.516} C_VEL
LIN {X 0,Y 333.652,Z 1243.93,A -85,B 0,C 180,E1 13423.065,E2 13423.065} C_VEL
LIN {X 0,Y 336.803,Z 1230.692,A -85,B 0,C 180,E1 13429.215,E2 13429.215} C_VEL
LIN {X 0,Y 342.035,Z 1212.07,A -85,B 0,C 180,E1 13434.962,E2 13434.962} C_VEL
LIN {X 0,Y 348.712,Z 1189.314,A -85,B 0,C 180,E1 13439.91,E2 13439.91} C_VEL
LIN {X 0,Y 356.2,Z 1162.274,A -85,B 0,C 180,E1 13444.141,E2 13444.141} C_VEL
LIN {X 0,Y 363.888,Z 1129.815,A -85,B 0,C 180,E1 13447.73,E2 13447.73} C_VEL
LIN {X 0,Y 370.265,Z 1095.404,A -85,B 0,C 180,E1 13450.31,E2 13450.31} C_VEL
LIN {X 0,Y 372.803,Z 1071.378,A -85,B 0,C 180,E1 13451.655,E2 13451.655} C_VEL
LIN {X 0,Y 360.113,Z 1041.297,A -85,B 0,C 180,E1 13454.999,E2 13454.999} C_VEL
LIN {X 0,Y 342.835,Z 1011.267,A -85,B 0,C 180,E1 13458.992,E2 13458.992} C_VEL
LIN {X 0,Y 331.924,Z 994.801,A -85,B 0,C 180,E1 13461.811,E2 13461.811} C_VEL
LIN {X 0,Y 329.494,Z 990.145,A -85,B 0,C 180,E1 13462.526,E2 13462.526} C_VEL
LIN {X 0,Y 329.413,Z 989.03,A -85,B 0,C 180,E1 13462.602,E2 13462.602} C_VEL
LIN {X 0,Y 329.648,Z 989.03,A -85,B 0,C 180,E1 13470.422,E2 13470.422} C_VEL
LIN {X 0,Y 329.989,Z 989.03,A -85,B 0,C 180,E1 13478.543,E2 13478.543} C_VEL
LIN {X 0,Y 330.357,Z 989.03,A -85,B 0,C 180,E1 13484.095,E2 13484.095} C_VEL
LIN {X 0,Y 330.806,Z 989.03,A -85,B 0,C 180,E1 13492.135,E2 13492.135} C_VEL
LIN {X 0,Y 331.345,Z 989.03,A -85,B 0,C 180,E1 13500.001,E2 13500.001} C_VEL
LIN {X 0,Y 330.779,Z 989.03,A -85,B 0,C 180,E1 13507.866,E2 13507.866} C_VEL
LIN {X 0,Y 330.259,Z 989.03,A -85,B 0,C 180,E1 13515.911,E2 13515.911} C_VEL
LIN {X 0,Y 329.826,Z 989.03,A -85,B 0,C 180,E1 13524.315,E2 13524.315} C_VEL
LIN {X 0,Y 329.588,Z 989.03,A -85,B 0,C 180,E1 13530.24,E2 13530.24} C_VEL
LIN {X 0,Y 329.662,Z 989.551,A -85,B 0,C 180,E1 13533.727,E2 13533.727} C_VEL
LIN {X 0,Y 334.303,Z 1001.24,A -85,B 0,C 180,E1 13535.41,E2 13535.41} C_VEL
LIN {X 0,Y 358.847,Z 1052.656,A -85,B 0,C 180,E1 13540.836,E2 13540.836} C_VEL
LIN {X 0,Y 372.168,Z 1087.791,A -85,B 0,C 180,E1 13544.297,E2 13544.297} C_VEL
LIN {X 0,Y 365.238,Z 1128.943,A -85,B 0,C 180,E1 13546.825,E2 13546.825} C_VEL
LIN {X 0,Y 357.193,Z 1166.788,A -85,B 0,C 180,E1 13550.172,E2 13550.172} C_VEL
LIN {X 0,Y 348.818,Z 1204.861,A -85,B 0,C 180,E1 13554.843,E2 13554.843} C_VEL
LIN {X 0,Y 342.846,Z 1233.716,A -85,B 0,C 180,E1 13559.339,E2 13559.339} C_VEL
LIN {X 0,Y 337.891,Z 1258.275,A -85,B 0,C 180,E1 13564.547,E2 13564.547} C_VEL
LIN {X 0,Y 334.369,Z 1277.816,A -85,B 0,C 180,E1 13570.221,E2 13570.221} C_VEL
LIN {X 0,Y 332.513,Z 1292.249,A -85,B 0,C 180,E1 13576.221,E2 13576.221} C_VEL
LIN {X 0,Y 331.89,Z 1301.207,A -85,B 0,C 180,E1 13582.165,E2 13582.165} C_VEL
LIN {X 0,Y 331.771,Z 1304.954,A -85,B 0,C 180,E1 13587.398,E2 13587.398} C_VEL
LIN {X 0,Y 331.815,Z 1304.955,A -85,B 0,C 180,E1 13592.612,E2 13592.612} C_VEL
LIN {X 0,Y 331.912,Z 1301.203,A -85,B 0,C 180,E1 13597.844,E2 13597.844} C_VEL
LIN {X 0,Y 332.57,Z 1292.236,A -85,B 0,C 180,E1 13603.787,E2 13603.787} C_VEL
LIN {X 0,Y 334.631,Z 1276.798,A -85,B 0,C 180,E1 13610.117,E2 13610.117} C_VEL
LIN {X 0,Y 338.361,Z 1256.907,A -85,B 0,C 180,E1 13615.781,E2 13615.781} C_VEL
LIN {X 0,Y 340.556,Z 1246.238,A -85,B 0,C 180,E1 13618.207,E2 13618.207} C_VEL
LIN {X 0,Y 339.24,Z 1235.72,A -85,B 0,C 180,E1 13620.56,E2 13620.56} C_VEL
LIN {X 0,Y 337.867,Z 1226.105,A -85,B 0,C 180,E1 13622.582,E2 13622.582} C_VEL
LIN {X 0,Y 338.144,Z 1224.571,A -85,B 0,C 180,E1 13622.848,E2 13622.848} C_VEL
LIN {X 0,Y 344.778,Z 1194.078,A -85,B 0,C 180,E1 13627.203,E2 13627.203} C_VEL
LIN {X 0,Y 351.069,Z 1159.772,A -85,B 0,C 180,E1 13630.681,E2 13630.681} C_VEL
LIN {X 0,Y 356.587,Z 1126.599,A -85,B 0,C 180,E1 13633.274,E2 13633.274} C_VEL
LIN {X 0,Y 366.039,Z 1087.737,A -85,B 0,C 180,E1 13636.374,E2 13636.374} C_VEL
LIN {X 0,Y 367.987,Z 1060.553,A -85,B 0,C 180,E1 13639.914,E2 13639.914} C_VEL
LIN {X 0,Y 366.822,Z 1056.151,A -85,B 0,C 180,E1 13641.9,E2 13641.9} C_VEL
LIN {X 0,Y 366.219,Z 1057.584,A -85,B 0,C 180,E1 13644.771,E2 13644.771} C_VEL
LIN {X 0,Y 365.696,Z 1061.414,A -85,B 0,C 180,E1 13645.654,E2 13645.654} C_VEL
LIN {X 0,Y 356.096,Z 1099.147,A -85,B 0,C 180,E1 13648.532,E2 13648.532} C_VEL
LIN {X 0,Y 349.386,Z 1127.562,A -85,B 0,C 180,E1 13651.635,E2 13651.635} C_VEL
LIN {X 0,Y 342.693,Z 1151.363,A -85,B 0,C 180,E1 13655.484,E2 13655.484} C_VEL
LIN {X 0,Y 336.805,Z 1169.768,A -85,B 0,C 180,E1 13659.865,E2 13659.865} C_VEL
LIN {X 0,Y 331.857,Z 1183.432,A -85,B 0,C 180,E1 13664.843,E2 13664.843} C_VEL
LIN {X 0,Y 328.977,Z 1190.968,A -85,B 0,C 180,E1 13669.428,E2 13669.428} C_VEL
LIN {X 0,Y 327.097,Z 1194.748,A -85,B 0,C 180,E1 13674.706,E2 13674.706} C_VEL
LIN {X 0,Y 326.439,Z 1193.653,A -85,B 0,C 180,E1 13679.999,E2 13679.999} C_VEL
LIN {X 0,Y 326.605,Z 1187.638,A -85,B 0,C 180,E1 13685.301,E2 13685.301} C_VEL
